LIN {X 0,Y 467.698,Z 216.222,A -85,B 0,C 180,E1 -7463.962,E2 -7463.962} C_VEL
LIN {X 0,Y 467.802,Z 216.212,A -85,B 0,C 180,E1 -7467.417,E2 -7467.417} C_VEL
LIN {X 0,Y 467.814,Z 216.207,A -85,B 0,C 180,E1 -7470,E2 -7470} C_VEL
LIN {X 0,Y 467.802,Z 216.211,A -85,B 0,C 180,E1 -7472.583,E2 -7472.583} C_VEL
LIN {X 0,Y 467.698,Z 216.222,A -85,B 0,C 180,E1 -7476.038,E2 -7476.038} C_VEL
LIN {X 0,Y 467.633,Z 216.235,A -85,B 0,C 180,E1 -7478.643,E2 -7478.643} C_VEL
LIN {X 0,Y 467.672,Z 216.264,A -85,B 0,C 180,E1 -7482.09,E2 -7482.09} C_VEL
LIN {X 0,Y 468.717,Z 223.503,A -85,B 0,C 180,E1 -7483.659,E2 -7483.659} C_VEL
LIN {X 0,Y 468.443,Z 235.17,A -85,B 0,C 180,E1 -7486.063,E2 -7486.063} C_VEL
LIN {X 0,Y 471.362,Z 250.846,A -85,B 0,C 180,E1 -7486.427,E2 -7486.427} C_VEL
LIN {X 0,Y 470.517,Z 341.953,A -85,B 0,C 180,E1 -7487.858,E2 -7487.858} C_VEL
LIN {X 0,Y 470.242,Z 355.17,A -85,B 0,C 180,E1 -7488.235,E2 -7488.235} C_VEL
LIN {X 0,Y 469.903,Z 367.496,A -85,B 0,C 180,E1 -7488.757,E2 -7488.757} C_VEL
LIN {X 0,Y 469.518,Z 379.697,A -85,B 0,C 180,E1 -7489.46,E2 -7489.46} C_VEL
LIN {X 0,Y 469.025,Z 390.638,A -85,B 0,C 180,E1 -7490.273,E2 -7490.273} C_VEL
LIN {X 0,Y 468.536,Z 401.021,A -85,B 0,C 180,E1 -7491.237,E2 -7491.237} C_VEL
LIN {X 0,Y 468.092,Z 410.16,A -85,B 0,C 180,E1 -7492.278,E2 -7492.278} C_VEL
LIN {X 0,Y 467.664,Z 419.305,A -85,B 0,C 180,E1 -7493.572,E2 -7493.572} C_VEL
LIN {X 0,Y 467.295,Z 426.861,A -85,B 0,C 180,E1 -7494.904,E2 -7494.904} C_VEL
LIN {X 0,Y 467.014,Z 433.368,A -85,B 0,C 180,E1 -7496.355,E2 -7496.355} C_VEL
LIN {X 0,Y 466.823,Z 438.356,A -85,B 0,C 180,E1 -7497.82,E2 -7497.82} C_VEL
LIN {X 0,Y 466.725,Z 441.75,A -85,B 0,C 180,E1 -7499.163,E2 -7499.163} C_VEL
LIN {X 0,Y 466.568,Z 444.553,A -85,B 0,C 180,E1 -7500.855,E2 -7500.855} C_VEL
LIN {X 0,Y 466.525,Z 445.764,A -85,B 0,C 180,E1 -7502.491,E2 -7502.491} C_VEL
LIN {X 0,Y 466.515,Z 445.58,A -85,B 0,C 180,E1 -7504.062,E2 -7504.062} C_VEL
LIN {X 0,Y 466.566,Z 444.162,A -85,B 0,C 180,E1 -7505.582,E2 -7505.582} C_VEL
LIN {X 0,Y 466.714,Z 441.569,A -85,B 0,C 180,E1 -7507.064,E2 -7507.064} C_VEL
LIN {X 0,Y 466.883,Z 437.838,A -85,B 0,C 180,E1 -7508.498,E2 -7508.498} C_VEL
LIN {X 0,Y 467.075,Z 432.923,A -85,B 0,C 180,E1 -7509.892,E2 -7509.892} C_VEL
LIN {X 0,Y 467.372,Z 425.882,A -85,B 0,C 180,E1 -7511.424,E2 -7511.424} C_VEL
LIN {X 0,Y 467.654,Z 419.182,A -85,B 0,C 180,E1 -7512.587,E2 -7512.587} C_VEL
LIN {X 0,Y 468.1,Z 411.54,A -85,B 0,C 180,E1 -7513.679,E2 -7513.679} C_VEL
LIN {X 0,Y 468.582,Z 401.758,A -85,B 0,C 180,E1 -7514.822,E2 -7514.822} C_VEL
LIN {X 0,Y 469.08,Z 390.527,A -85,B 0,C 180,E1 -7515.87,E2 -7515.87} C_VEL
LIN {X 0,Y 469.594,Z 379.793,A -85,B 0,C 180,E1 -7516.666,E2 -7516.666} C_VEL
LIN {X 0,Y 470.011,Z 367.432,A -85,B 0,C 180,E1 -7517.375,E2 -7517.375} C_VEL
LIN {X 0,Y 470.382,Z 354.341,A -85,B 0,C 180,E1 -7517.921,E2 -7517.921} C_VEL
LIN {X 0,Y 470.62,Z 341.699,A -85,B 0,C 180,E1 -7518.271,E2 -7518.271} C_VEL
LIN {X 0,Y 471.439,Z 249.982,A -85,B 0,C 180,E1 -7519.719,E2 -7519.719} C_VEL
LIN {X 0,Y 468.517,Z 235.14,A -85,B 0,C 180,E1 -7520.078,E2 -7520.078} C_VEL
LIN {X 0,Y 468.684,Z 222.897,A -85,B 0,C 180,E1 -7522.429,E2 -7522.429} C_VEL
LIN {X 0,Y 467.576,Z 216.244,A -85,B 0,C 180,E1 -7523.788,E2 -7523.788} C_VEL
LIN {X 0,Y 467.548,Z 216.245,A -85,B 0,C 180,E1 -7526.217,E2 -7526.217} C_VEL
LIN {X 0,Y 467.538,Z 216.249,A -85,B 0,C 180,E1 -7529.272,E2 -7529.272} C_VEL
LIN {X 0,Y 467.611,Z 216.236,A -85,B 0,C 180,E1 -7532.464,E2 -7532.464} C_VEL
LIN {X 0,Y 467.572,Z 216.245,A -85,B 0,C 180,E1 -7535.118,E2 -7535.118} C_VEL
LIN {X 0,Y 467.505,Z 216.247,A -85,B 0,C 180,E1 -7537.931,E2 -7537.931} C_VEL
LIN {X 0,Y 467.596,Z 216.24,A -85,B 0,C 180,E1 -7540.697,E2 -7540.697} C_VEL
LIN {X 0,Y 467.625,Z 216.234,A -85,B 0,C 180,E1 -7544.12,E2 -7544.12} C_VEL
LIN {X 0,Y 467.662,Z 216.227,A -85,B 0,C 180,E1 -7547.86,E2 -7547.86} C_VEL
LIN {X 0,Y 467.652,Z 216.229,A -85,B 0,C 180,E1 -7551.362,E2 -7551.362} C_VEL
LIN {X 0,Y 467.713,Z 216.221,A -85,B 0,C 180,E1 -7553.967,E2 -7553.967} C_VEL
LIN {X 0,Y 467.841,Z 216.204,A -85,B 0,C 180,E1 -7557.422,E2 -7557.422} C_VEL
LIN {X 0,Y 467.865,Z 216.202,A -85,B 0,C 180,E1 -7560.005,E2 -7560.005} C_VEL
LIN {X 0,Y 467.809,Z 216.211,A -85,B 0,C 180,E1 -7562.588,E2 -7562.588} C_VEL
LIN {X 0,Y 467.713,Z 216.218,A -85,B 0,C 180,E1 -7566.042,E2 -7566.042} C_VEL
LIN {X 0,Y 467.653,Z 216.234,A -85,B 0,C 180,E1 -7568.648,E2 -7568.648} C_VEL
LIN {X 0,Y 467.65,Z 216.23,A -85,B 0,C 180,E1 -7572.15,E2 -7572.15} C_VEL
LIN {X 0,Y 467.635,Z 216.23,A -85,B 0,C 180,E1 -7575.699,E2 -7575.699} C_VEL
LIN {X 0,Y 467.619,Z 216.232,A -85,B 0,C 180,E1 -7579.312,E2 -7579.312} C_VEL
LIN {X 0,Y 467.53,Z 216.244,A -85,B 0,C 180,E1 -7582.078,E2 -7582.078} C_VEL
LIN {X 0,Y 467.549,Z 216.243,A -85,B 0,C 180,E1 -7584.894,E2 -7584.894} C_VEL
LIN {X 0,Y 467.547,Z 216.241,A -85,B 0,C 180,E1 -7587.777,E2 -7587.777} C_VEL
LIN {X 0,Y 467.548,Z 216.243,A -85,B 0,C 180,E1 -7591.043,E2 -7591.043} C_VEL
LIN {X 0,Y 467.578,Z 216.24,A -85,B 0,C 180,E1 -7594.243,E2 -7594.243} C_VEL
LIN {X 0,Y 467.517,Z 216.245,A -85,B 0,C 180,E1 -7597.183,E2 -7597.183} C_VEL
LIN {X 0,Y 467.522,Z 216.249,A -85,B 0,C 180,E1 -7600.274,E2 -7600.274} C_VEL
LIN {X 0,Y 467.522,Z 216.251,A -85,B 0,C 180,E1 -7602.571,E2 -7602.571} C_VEL
LIN {X 0,Y 467.558,Z 216.243,A -85,B 0,C 180,E1 -7605.053,E2 -7605.053} C_VEL
LIN {X 0,Y 467.556,Z 216.244,A -85,B 0,C 180,E1 -7608.73,E2 -7608.73} C_VEL
LIN {X 0,Y 467.539,Z 216.247,A -85,B 0,C 180,E1 -7611.954,E2 -7611.954} C_VEL
LIN {X 0,Y 467.545,Z 216.243,A -85,B 0,C 180,E1 -7615.167,E2 -7615.167} C_VEL
LIN {X 0,Y 467.549,Z 216.252,A -85,B 0,C 180,E1 -7618.258,E2 -7618.258} C_VEL
LIN {X 0,Y 467.526,Z 216.249,A -85,B 0,C 180,E1 -7621.248,E2 -7621.248} C_VEL
LIN {X 0,Y 467.563,Z 216.308,A -85,B 0,C 180,E1 -7624.098,E2 -7624.098} C_VEL
LIN {X 0,Y 469.703,Z 227.399,A -85,B 0,C 180,E1 -7626.173,E2 -7626.173} C_VEL
LIN {X 0,Y 469.196,Z 242.28,A -85,B 0,C 180,E1 -7628.742,E2 -7628.742} C_VEL
LIN {X 0,Y 468.518,Z 260.61,A -85,B 0,C 180,E1 -7631.865,E2 -7631.865} C_VEL
LIN {X 0,Y 468.314,Z 267.311,A -85,B 0,C 180,E1 -7632.96,E2 -7632.96} C_VEL
LIN {X 0,Y 471.186,Z 286.372,A -85,B 0,C 180,E1 -7633.375,E2 -7633.375} C_VEL
LIN {X 0,Y 470.504,Z 375.82,A -85,B 0,C 180,E1 -7634.792,E2 -7634.792} C_VEL
LIN {X 0,Y 470.072,Z 389.744,A -85,B 0,C 180,E1 -7635.193,E2 -7635.193} C_VEL
LIN {X 0,Y 469.595,Z 402.758,A -85,B 0,C 180,E1 -7635.759,E2 -7635.759} C_VEL
LIN {X 0,Y 469.093,Z 414.583,A -85,B 0,C 180,E1 -7636.462,E2 -7636.462} C_VEL
LIN {X 0,Y 468.57,Z 426.698,A -85,B 0,C 180,E1 -7637.389,E2 -7637.389} C_VEL
LIN {X 0,Y 468.149,Z 436.288,A -85,B 0,C 180,E1 -7638.307,E2 -7638.307} C_VEL
LIN {X 0,Y 467.672,Z 445.54,A -85,B 0,C 180,E1 -7639.392,E2 -7639.392} C_VEL
LIN {X 0,Y 467.253,Z 454.552,A -85,B 0,C 180,E1 -7640.695,E2 -7640.695} C_VEL
LIN {X 0,Y 467.003,Z 461.815,A -85,B 0,C 180,E1 -7641.998,E2 -7641.998} C_VEL
LIN {X 0,Y 466.839,Z 466.717,A -85,B 0,C 180,E1 -7643.083,E2 -7643.083} C_VEL
LIN {X 0,Y 466.736,Z 471.485,A -85,B 0,C 180,E1 -7644.383,E2 -7644.383} C_VEL
LIN {X 0,Y 466.649,Z 475.131,A -85,B 0,C 180,E1 -7645.682,E2 -7645.682} C_VEL
LIN {X 0,Y 466.693,Z 477.016,A -85,B 0,C 180,E1 -7646.547,E2 -7646.547} C_VEL
LIN {X 0,Y 466.666,Z 478.428,A -85,B 0,C 180,E1 -7647.411,E2 -7647.411} C_VEL
LIN {X 0,Y 466.624,Z 480.056,A -85,B 0,C 180,E1 -7649.137,E2 -7649.137} C_VEL
LIN {X 0,Y 466.606,Z 480.277,A -85,B 0,C 180,E1 -7650,E2 -7650} C_VEL
LIN {X 0,Y 466.624,Z 480.063,A -85,B 0,C 180,E1 -7650.863,E2 -7650.863} C_VEL
LIN {X 0,Y 466.666,Z 478.457,A -85,B 0,C 180,E1 -7652.589,E2 -7652.589} C_VEL
LIN {X 0,Y 466.693,Z 477.051,A -85,B 0,C 180,E1 -7653.453,E2 -7653.453} C_VEL
LIN {X 0,Y 466.691,Z 474.094,A -85,B 0,C 180,E1 -7654.751,E2 -7654.751} C_VEL
LIN {X 0,Y 466.747,Z 470.089,A -85,B 0,C 180,E1 -7656.05,E2 -7656.05} C_VEL
LIN {X 0,Y 466.926,Z 463.923,A -85,B 0,C 180,E1 -7657.568,E2 -7657.568} C_VEL
LIN {X 0,Y 467.166,Z 457.189,A -85,B 0,C 180,E1 -7658.87,E2 -7658.87} C_VEL
LIN {X 0,Y 467.493,Z 448.832,A -85,B 0,C 180,E1 -7660.174,E2 -7660.174} C_VEL
LIN {X 0,Y 467.955,Z 440.241,A -85,B 0,C 180,E1 -7661.259,E2 -7661.259} C_VEL
LIN {X 0,Y 468.445,Z 430.165,A -85,B 0,C 180,E1 -7662.295,E2 -7662.295} C_VEL
LIN {X 0,Y 468.881,Z 419.128,A -85,B 0,C 180,E1 -7663.213,E2 -7663.213} C_VEL
LIN {X 0,Y 469.377,Z 407.552,A -85,B 0,C 180,E1 -7663.971,E2 -7663.971} C_VEL
LIN {X 0,Y 469.837,Z 395.543,A -85,B 0,C 180,E1 -7664.565,E2 -7664.565} C_VEL
LIN {X 0,Y 470.253,Z 382.567,A -85,B 0,C 180,E1 -7665.023,E2 -7665.023} C_VEL
LIN {X 0,Y 470.538,Z 368.731,A -85,B 0,C 180,E1 -7665.318,E2 -7665.318} C_VEL
LIN {X 0,Y 471.01,Z 285.555,A -85,B 0,C 180,E1 -7666.617,E2 -7666.617} C_VEL
LIN {X 0,Y 468.273,Z 267.515,A -85,B 0,C 180,E1 -7667.017,E2 -7667.017} C_VEL
LIN {X 0,Y 468.932,Z 250.577,A -85,B 0,C 180,E1 -7669.935,E2 -7669.935} C_VEL
LIN {X 0,Y 469.674,Z 234.928,A -85,B 0,C 180,E1 -7672.663,E2 -7672.663} C_VEL
LIN {X 0,Y 469.875,Z 228.39,A -85,B 0,C 180,E1 -7673.818,E2 -7673.818} C_VEL
LIN {X 0,Y 467.555,Z 216.246,A -85,B 0,C 180,E1 -7676.142,E2 -7676.142} C_VEL
LIN {X 0,Y 467.532,Z 216.249,A -85,B 0,C 180,E1 -7679.32,E2 -7679.32} C_VEL
LIN {X 0,Y 467.545,Z 216.248,A -85,B 0,C 180,E1 -7681.742,E2 -7681.742} C_VEL
LIN {X 0,Y 467.518,Z 216.244,A -85,B 0,C 180,E1 -7684.836,E2 -7684.836} C_VEL
LIN {X 0,Y 467.537,Z 216.246,A -85,B 0,C 180,E1 -7688.046,E2 -7688.046} C_VEL
LIN {X 0,Y 467.553,Z 216.243,A -85,B 0,C 180,E1 -7691.404,E2 -7691.404} C_VEL
LIN {X 0,Y 467.535,Z 216.243,A -85,B 0,C 180,E1 -7695.045,E2 -7695.045} C_VEL
LIN {X 0,Y 467.554,Z 216.24,A -85,B 0,C 180,E1 -7698.591,E2 -7698.591} C_VEL
LIN {X 0,Y 467.533,Z 216.247,A -85,B 0,C 180,E1 -7701.949,E2 -7701.949} C_VEL
LIN {X 0,Y 467.518,Z 216.246,A -85,B 0,C 180,E1 -7705.16,E2 -7705.16} C_VEL
LIN {X 0,Y 467.544,Z 216.242,A -85,B 0,C 180,E1 -7708.253,E2 -7708.253} C_VEL
LIN {X 0,Y 467.52,Z 216.247,A -85,B 0,C 180,E1 -7711.243,E2 -7711.243} C_VEL
LIN {X 0,Y 467.558,Z 216.24,A -85,B 0,C 180,E1 -7714.403,E2 -7714.403} C_VEL
LIN {X 0,Y 467.571,Z 216.239,A -85,B 0,C 180,E1 -7716.992,E2 -7716.992} C_VEL
LIN {X 0,Y 467.589,Z 216.241,A -85,B 0,C 180,E1 -7719.772,E2 -7719.772} C_VEL
LIN {X 0,Y 467.568,Z 216.238,A -85,B 0,C 180,E1 -7722.501,E2 -7722.501} C_VEL
LIN {X 0,Y 467.589,Z 216.238,A -85,B 0,C 180,E1 -7725.192,E2 -7725.192} C_VEL
LIN {X 0,Y 467.629,Z 216.235,A -85,B 0,C 180,E1 -7727.85,E2 -7727.85} C_VEL
LIN {X 0,Y 467.621,Z 216.237,A -85,B 0,C 180,E1 -7731.352,E2 -7731.352} C_VEL
LIN {X 0,Y 467.692,Z 216.225,A -85,B 0,C 180,E1 -7733.957,E2 -7733.957} C_VEL
LIN {X 0,Y 467.777,Z 216.219,A -85,B 0,C 180,E1 -7737.412,E2 -7737.412} C_VEL
LIN {X 0,Y 467.833,Z 216.207,A -85,B 0,C 180,E1 -7739.995,E2 -7739.995} C_VEL
LIN {X 0,Y 467.806,Z 216.208,A -85,B 0,C 180,E1 -7742.578,E2 -7742.578} C_VEL
LIN {X 0,Y 467.675,Z 216.226,A -85,B 0,C 180,E1 -7746.033,E2 -7746.033} C_VEL
LIN {X 0,Y 467.616,Z 216.232,A -85,B 0,C 180,E1 -7748.639,E2 -7748.639} C_VEL
LIN {X 0,Y 467.634,Z 216.23,A -85,B 0,C 180,E1 -7752.14,E2 -7752.14} C_VEL
LIN {X 0,Y 467.624,Z 216.233,A -85,B 0,C 180,E1 -7755.879,E2 -7755.879} C_VEL
LIN {X 0,Y 467.594,Z 216.242,A -85,B 0,C 180,E1 -7759.303,E2 -7759.303} C_VEL
LIN {X 0,Y 467.501,Z 216.247,A -85,B 0,C 180,E1 -7762.069,E2 -7762.069} C_VEL
LIN {X 0,Y 467.536,Z 216.244,A -85,B 0,C 180,E1 -7764.884,E2 -7764.884} C_VEL
LIN {X 0,Y 467.581,Z 216.239,A -85,B 0,C 180,E1 -7767.764,E2 -7767.764} C_VEL
LIN {X 0,Y 467.53,Z 216.247,A -85,B 0,C 180,E1 -7771.039,E2 -7771.039} C_VEL
LIN {X 0,Y 467.548,Z 216.24,A -85,B 0,C 180,E1 -7774.237,E2 -7774.237} C_VEL
LIN {X 0,Y 467.505,Z 216.252,A -85,B 0,C 180,E1 -7777.181,E2 -7777.181} C_VEL
LIN {X 0,Y 467.533,Z 216.242,A -85,B 0,C 180,E1 -7780.26,E2 -7780.26} C_VEL
LIN {X 0,Y 467.541,Z 216.242,A -85,B 0,C 180,E1 -7782.562,E2 -7782.562} C_VEL
LIN {X 0,Y 467.522,Z 216.249,A -85,B 0,C 180,E1 -7785.049,E2 -7785.049} C_VEL
LIN {X 0,Y 467.539,Z 216.247,A -85,B 0,C 180,E1 -7787.436,E2 -7787.436} C_VEL
LIN {X 0,Y 467.53,Z 216.246,A -85,B 0,C 180,E1 -7790.851,E2 -7790.851} C_VEL
LIN {X 0,Y 467.51,Z 216.245,A -85,B 0,C 180,E1 -7794.256,E2 -7794.256} C_VEL
LIN {X 0,Y 467.526,Z 216.25,A -85,B 0,C 180,E1 -7797.317,E2 -7797.317} C_VEL
LIN {X 0,Y 467.519,Z 216.246,A -85,B 0,C 180,E1 -7800.663,E2 -7800.663} C_VEL
LIN {X 0,Y 467.561,Z 216.247,A -85,B 0,C 180,E1 -7803.197,E2 -7803.197} C_VEL
LIN {X 0,Y 467.526,Z 216.243,A -85,B 0,C 180,E1 -7806.055,E2 -7806.055} C_VEL
LIN {X 0,Y 467.579,Z 216.241,A -85,B 0,C 180,E1 -7808.855,E2 -7808.855} C_VEL
LIN {X 0,Y 467.578,Z 216.239,A -85,B 0,C 180,E1 -7811.613,E2 -7811.613} C_VEL
LIN {X 0,Y 467.591,Z 216.235,A -85,B 0,C 180,E1 -7814.304,E2 -7814.304} C_VEL
LIN {X 0,Y 467.536,Z 216.247,A -85,B 0,C 180,E1 -7815.371,E2 -7815.371} C_VEL
LIN {X 0,Y 466.869,Z 216.326,A -85,B 0,C 180,E1 -7816.091,E2 -7816.091} C_VEL
LIN {X 0,Y 464.039,Z 216.684,A -85,B 0,C 180,E1 -7817.26,E2 -7817.26} C_VEL
LIN {X 0,Y 461.647,Z 216.978,A -85,B 0,C 180,E1 -7818.203,E2 -7818.203} C_VEL
LIN {X 0,Y 460.618,Z 217.11,A -85,B 0,C 180,E1 -7818.931,E2 -7818.931} C_VEL
LIN {X 0,Y 460.533,Z 217.116,A -85,B 0,C 180,E1 -7819.177,E2 -7819.177} C_VEL
LIN {X 0,Y 460.665,Z 217.1,A -85,B 0,C 180,E1 -7822.527,E2 -7822.527} C_VEL
LIN {X 0,Y 460.644,Z 217.104,A -85,B 0,C 180,E1 -7824.748,E2 -7824.748} C_VEL
LIN {X 0,Y 460.768,Z 217.089,A -85,B 0,C 180,E1 -7827.377,E2 -7827.377} C_VEL
LIN {X 0,Y 460.786,Z 217.083,A -85,B 0,C 180,E1 -7830,E2 -7830} C_VEL
LIN {X 0,Y 460.768,Z 217.088,A -85,B 0,C 180,E1 -7832.623,E2 -7832.623} C_VEL
LIN {X 0,Y 460.664,Z 217.098,A -85,B 0,C 180,E1 -7836.13,E2 -7836.13} C_VEL
LIN {X 0,Y 460.6,Z 217.113,A -85,B 0,C 180,E1 -7838.776,E2 -7838.776} C_VEL
LIN {X 0,Y 460.656,Z 217.258,A -85,B 0,C 180,E1 -7841.941,E2 -7841.941} C_VEL
LIN {X 0,Y 461.758,Z 225.024,A -85,B 0,C 180,E1 -7843.645,E2 -7843.645} C_VEL
LIN {X 0,Y 461.495,Z 235.327,A -85,B 0,C 180,E1 -7845.796,E2 -7845.796} C_VEL
LIN {X 0,Y 464.529,Z 250.64,A -85,B 0,C 180,E1 -7846.175,E2 -7846.175} C_VEL
LIN {X 0,Y 463.66,Z 342.57,A -85,B 0,C 180,E1 -7847.647,E2 -7847.647} C_VEL
LIN {X 0,Y 463.364,Z 355.678,A -85,B 0,C 180,E1 -7848.029,E2 -7848.029} C_VEL
LIN {X 0,Y 463.007,Z 368.52,A -85,B 0,C 180,E1 -7848.587,E2 -7848.587} C_VEL
LIN {X 0,Y 462.595,Z 380.416,A -85,B 0,C 180,E1 -7849.295,E2 -7849.295} C_VEL
LIN {X 0,Y 462.023,Z 392.472,A -85,B 0,C 180,E1 -7850.223,E2 -7850.223} C_VEL
LIN {X 0,Y 461.497,Z 402.613,A -85,B 0,C 180,E1 -7851.203,E2 -7851.203} C_VEL
LIN {X 0,Y 460.961,Z 412.559,A -85,B 0,C 180,E1 -7852.405,E2 -7852.405} C_VEL
LIN {X 0,Y 460.527,Z 421.341,A -85,B 0,C 180,E1 -7853.723,E2 -7853.723} C_VEL
LIN {X 0,Y 460.239,Z 428.51,A -85,B 0,C 180,E1 -7855.071,E2 -7855.071} C_VEL
LIN {X 0,Y 459.943,Z 433.788,A -85,B 0,C 180,E1 -7856.303,E2 -7856.303} C_VEL
LIN {X 0,Y 459.789,Z 438.129,A -85,B 0,C 180,E1 -7857.575,E2 -7857.575} C_VEL
LIN {X 0,Y 459.676,Z 441.325,A -85,B 0,C 180,E1 -7858.789,E2 -7858.789} C_VEL
LIN {X 0,Y 459.5,Z 444.151,A -85,B 0,C 180,E1 -7860.313,E2 -7860.313} C_VEL
LIN {X 0,Y 459.457,Z 445.324,A -85,B 0,C 180,E1 -7861.336,E2 -7861.336} C_VEL
LIN {X 0,Y 459.411,Z 446.073,A -85,B 0,C 180,E1 -7862.728,E2 -7862.728} C_VEL
LIN {X 0,Y 459.432,Z 445.628,A -85,B 0,C 180,E1 -7864.47,E2 -7864.47} C_VEL
LIN {X 0,Y 459.511,Z 444.126,A -85,B 0,C 180,E1 -7865.858,E2 -7865.858} C_VEL
LIN {X 0,Y 459.672,Z 441.336,A -85,B 0,C 180,E1 -7867.354,E2 -7867.354} C_VEL
LIN {X 0,Y 459.838,Z 437.42,A -85,B 0,C 180,E1 -7868.801,E2 -7868.801} C_VEL
LIN {X 0,Y 460.069,Z 432.327,A -85,B 0,C 180,E1 -7870.211,E2 -7870.211} C_VEL
LIN {X 0,Y 460.348,Z 425.988,A -85,B 0,C 180,E1 -7871.588,E2 -7871.588} C_VEL
LIN {X 0,Y 460.75,Z 418.144,A -85,B 0,C 180,E1 -7872.943,E2 -7872.943} C_VEL
LIN {X 0,Y 461.204,Z 409.879,A -85,B 0,C 180,E1 -7874.094,E2 -7874.094} C_VEL
LIN {X 0,Y 461.732,Z 400.209,A -85,B 0,C 180,E1 -7875.193,E2 -7875.193} C_VEL
LIN {X 0,Y 462.192,Z 390.615,A -85,B 0,C 180,E1 -7876.084,E2 -7876.084} C_VEL
LIN {X 0,Y 462.707,Z 379.833,A -85,B 0,C 180,E1 -7876.892,E2 -7876.892} C_VEL
LIN {X 0,Y 463.142,Z 367.848,A -85,B 0,C 180,E1 -7877.588,E2 -7877.588} C_VEL
LIN {X 0,Y 463.542,Z 354.862,A -85,B 0,C 180,E1 -7878.14,E2 -7878.14} C_VEL
LIN {X 0,Y 463.798,Z 341.73,A -85,B 0,C 180,E1 -7878.509,E2 -7878.509} C_VEL
LIN {X 0,Y 464.545,Z 250.039,A -85,B 0,C 180,E1 -7879.985,E2 -7879.985} C_VEL
LIN {X 0,Y 461.585,Z 235.343,A -85,B 0,C 180,E1 -7880.362,E2 -7880.362} C_VEL
LIN {X 0,Y 461.766,Z 224.266,A -85,B 0,C 180,E1 -7882.507,E2 -7882.507} C_VEL
LIN {X 0,Y 460.526,Z 217.122,A -85,B 0,C 180,E1 -7883.979,E2 -7883.979} C_VEL
LIN {X 0,Y 460.493,Z 217.128,A -85,B 0,C 180,E1 -7887.075,E2 -7887.075} C_VEL
LIN {X 0,Y 460.512,Z 217.122,A -85,B 0,C 180,E1 -7890.443,E2 -7890.443} C_VEL
LIN {X 0,Y 460.551,Z 217.118,A -85,B 0,C 180,E1 -7892.762,E2 -7892.762} C_VEL
LIN {X 0,Y 460.511,Z 217.12,A -85,B 0,C 180,E1 -7895.673,E2 -7895.673} C_VEL
LIN {X 0,Y 460.493,Z 217.124,A -85,B 0,C 180,E1 -7898.584,E2 -7898.584} C_VEL
LIN {X 0,Y 460.564,Z 217.117,A -85,B 0,C 180,E1 -7901.316,E2 -7901.316} C_VEL
LIN {X 0,Y 460.58,Z 217.111,A -85,B 0,C 180,E1 -7904.064,E2 -7904.064} C_VEL
LIN {X 0,Y 460.609,Z 217.106,A -85,B 0,C 180,E1 -7907.672,E2 -7907.672} C_VEL
LIN {X 0,Y 460.603,Z 217.108,A -85,B 0,C 180,E1 -7911.229,E2 -7911.229} C_VEL
LIN {X 0,Y 460.679,Z 217.097,A -85,B 0,C 180,E1 -7913.875,E2 -7913.875} C_VEL
LIN {X 0,Y 460.783,Z 217.084,A -85,B 0,C 180,E1 -7917.383,E2 -7917.383} C_VEL
LIN {X 0,Y 460.835,Z 217.078,A -85,B 0,C 180,E1 -7920.005,E2 -7920.005} C_VEL
LIN {X 0,Y 460.753,Z 217.09,A -85,B 0,C 180,E1 -7922.628,E2 -7922.628} C_VEL
LIN {X 0,Y 460.679,Z 217.095,A -85,B 0,C 180,E1 -7926.135,E2 -7926.135} C_VEL
LIN {X 0,Y 460.601,Z 217.11,A -85,B 0,C 180,E1 -7928.781,E2 -7928.781} C_VEL
LIN {X 0,Y 460.592,Z 217.113,A -85,B 0,C 180,E1 -7932.439,E2 -7932.439} C_VEL
LIN {X 0,Y 460.598,Z 217.108,A -85,B 0,C 180,E1 -7936.002,E2 -7936.002} C_VEL
LIN {X 0,Y 460.566,Z 217.11,A -85,B 0,C 180,E1 -7939.62,E2 -7939.62} C_VEL
LIN {X 0,Y 460.507,Z 217.121,A -85,B 0,C 180,E1 -7942.433,E2 -7942.433} C_VEL
LIN {X 0,Y 460.522,Z 217.116,A -85,B 0,C 180,E1 -7945.793,E2 -7945.793} C_VEL
LIN {X 0,Y 460.525,Z 217.115,A -85,B 0,C 180,E1 -7949.236,E2 -7949.236} C_VEL
LIN {X 0,Y 460.52,Z 217.122,A -85,B 0,C 180,E1 -7952.289,E2 -7952.289} C_VEL
LIN {X 0,Y 460.503,Z 217.119,A -85,B 0,C 180,E1 -7955.45,E2 -7955.45} C_VEL
LIN {X 0,Y 460.486,Z 217.123,A -85,B 0,C 180,E1 -7958.89,E2 -7958.89} C_VEL
LIN {X 0,Y 460.5,Z 217.121,A -85,B 0,C 180,E1 -7961.6,E2 -7961.6} C_VEL
LIN {X 0,Y 460.511,Z 217.124,A -85,B 0,C 180,E1 -7964.593,E2 -7964.593} C_VEL
LIN {X 0,Y 460.477,Z 217.126,A -85,B 0,C 180,E1 -7967.815,E2 -7967.815} C_VEL
LIN {X 0,Y 460.48,Z 217.129,A -85,B 0,C 180,E1 -7970.134,E2 -7970.134} C_VEL
LIN {X 0,Y 460.46,Z 217.126,A -85,B 0,C 180,E1 -7973.47,E2 -7973.47} C_VEL
LIN {X 0,Y 460.506,Z 217.124,A -85,B 0,C 180,E1 -7976.674,E2 -7976.674} C_VEL
LIN {X 0,Y 460.485,Z 217.129,A -85,B 0,C 180,E1 -7979.759,E2 -7979.759} C_VEL
LIN {X 0,Y 460.484,Z 217.126,A -85,B 0,C 180,E1 -7982.751,E2 -7982.751} C_VEL
LIN {X 0,Y 460.511,Z 217.136,A -85,B 0,C 180,E1 -7983.867,E2 -7983.867} C_VEL
LIN {X 0,Y 462.61,Z 227.87,A -85,B 0,C 180,E1 -7985.913,E2 -7985.913} C_VEL
LIN {X 0,Y 462.708,Z 232.485,A -85,B 0,C 180,E1 -7986.74,E2 -7986.74} C_VEL
LIN {X 0,Y 461.993,Z 248.444,A -85,B 0,C 180,E1 -7989.52,E2 -7989.52} C_VEL
LIN {X 0,Y 461.402,Z 264.339,A -85,B 0,C 180,E1 -7992.264,E2 -7992.264} C_VEL
LIN {X 0,Y 461.317,Z 266.734,A -85,B 0,C 180,E1 -7992.675,E2 -7992.675} C_VEL
LIN {X 0,Y 464.405,Z 287.188,A -85,B 0,C 180,E1 -7993.134,E2 -7993.134} C_VEL
LIN {X 0,Y 463.679,Z 375.696,A -85,B 0,C 180,E1 -7994.562,E2 -7994.562} C_VEL
LIN {X 0,Y 463.213,Z 389.565,A -85,B 0,C 180,E1 -7994.969,E2 -7994.969} C_VEL
LIN {X 0,Y 462.72,Z 402.546,A -85,B 0,C 180,E1 -7995.543,E2 -7995.543} C_VEL
LIN {X 0,Y 462.157,Z 414.355,A -85,B 0,C 180,E1 -7996.255,E2 -7996.255} C_VEL
LIN {X 0,Y 461.664,Z 425.832,A -85,B 0,C 180,E1 -7997.143,E2 -7997.143} C_VEL
LIN {X 0,Y 461.176,Z 436.039,A -85,B 0,C 180,E1 -7998.128,E2 -7998.128} C_VEL
LIN {X 0,Y 460.643,Z 445.284,A -85,B 0,C 180,E1 -7999.229,E2 -7999.229} C_VEL
LIN {X 0,Y 460.206,Z 454.294,A -85,B 0,C 180,E1 -8000.551,E2 -8000.551} C_VEL
LIN {X 0,Y 459.931,Z 461.556,A -85,B 0,C 180,E1 -8001.875,E2 -8001.875} C_VEL
LIN {X 0,Y 459.745,Z 467.64,A -85,B 0,C 180,E1 -8003.273,E2 -8003.273} C_VEL
LIN {X 0,Y 459.646,Z 472.554,A -85,B 0,C 180,E1 -8004.736,E2 -8004.736} C_VEL
LIN {X 0,Y 459.567,Z 474.873,A -85,B 0,C 180,E1 -8005.615,E2 -8005.615} C_VEL
LIN {X 0,Y 459.588,Z 476.756,A -85,B 0,C 180,E1 -8006.493,E2 -8006.493} C_VEL
LIN {X 0,Y 459.588,Z 478.169,A -85,B 0,C 180,E1 -8007.371,E2 -8007.371} C_VEL
LIN {X 0,Y 459.528,Z 479.795,A -85,B 0,C 180,E1 -8009.124,E2 -8009.124} C_VEL
LIN {X 0,Y 459.537,Z 480.016,A -85,B 0,C 180,E1 -8010,E2 -8010} C_VEL
LIN {X 0,Y 459.546,Z 479.19,A -85,B 0,C 180,E1 -8011.753,E2 -8011.753} C_VEL
LIN {X 0,Y 459.589,Z 478.191,A -85,B 0,C 180,E1 -8012.629,E2 -8012.629} C_VEL
LIN {X 0,Y 459.589,Z 476.78,A -85,B 0,C 180,E1 -8013.507,E2 -8013.507} C_VEL
LIN {X 0,Y 459.618,Z 473.82,A -85,B 0,C 180,E1 -8014.824,E2 -8014.824} C_VEL
LIN {X 0,Y 459.725,Z 468.764,A -85,B 0,C 180,E1 -8016.431,E2 -8016.431} C_VEL
LIN {X 0,Y 459.894,Z 462.615,A -85,B 0,C 180,E1 -8017.905,E2 -8017.905} C_VEL
LIN {X 0,Y 460.169,Z 455.643,A -85,B 0,C 180,E1 -8019.228,E2 -8019.228} C_VEL
LIN {X 0,Y 460.527,Z 446.899,A -85,B 0,C 180,E1 -8020.552,E2 -8020.552} C_VEL
LIN {X 0,Y 461.051,Z 437.948,A -85,B 0,C 180,E1 -8021.652,E2 -8021.652} C_VEL
LIN {X 0,Y 461.554,Z 427.263,A -85,B 0,C 180,E1 -8022.723,E2 -8022.723} C_VEL
LIN {X 0,Y 462.091,Z 415.709,A -85,B 0,C 180,E1 -8023.635,E2 -8023.635} C_VEL
LIN {X 0,Y 462.606,Z 403.161,A -85,B 0,C 180,E1 -8024.405,E2 -8024.405} C_VEL
LIN {X 0,Y 463.161,Z 390.339,A -85,B 0,C 180,E1 -8024.977,E2 -8024.977} C_VEL
LIN {X 0,Y 463.504,Z 376.681,A -85,B 0,C 180,E1 -8025.387,E2 -8025.387} C_VEL
LIN {X 0,Y 464.105,Z 323.215,A -85,B 0,C 180,E1 -8026.253,E2 -8026.253} C_VEL
LIN {X 0,Y 464.146,Z 285.68,A -85,B 0,C 180,E1 -8026.858,E2 -8026.858} C_VEL
LIN {X 0,Y 461.309,Z 267.29,A -85,B 0,C 180,E1 -8027.271,E2 -8027.271} C_VEL
LIN {X 0,Y 462.003,Z 250.301,A -85,B 0,C 180,E1 -8030.247,E2 -8030.247} C_VEL
LIN {X 0,Y 462.76,Z 234.639,A -85,B 0,C 180,E1 -8033.02,E2 -8033.02} C_VEL
LIN {X 0,Y 462.898,Z 229.408,A -85,B 0,C 180,E1 -8033.962,E2 -8033.962} C_VEL
LIN {X 0,Y 460.511,Z 217.124,A -85,B 0,C 180,E1 -8036.359,E2 -8036.359} C_VEL
LIN {X 0,Y 460.499,Z 217.125,A -85,B 0,C 180,E1 -8039.547,E2 -8039.547} C_VEL
LIN {X 0,Y 460.49,Z 217.122,A -85,B 0,C 180,E1 -8042.287,E2 -8042.287} C_VEL
LIN {X 0,Y 460.466,Z 217.126,A -85,B 0,C 180,E1 -8045.449,E2 -8045.449} C_VEL
LIN {X 0,Y 460.496,Z 217.119,A -85,B 0,C 180,E1 -8048.735,E2 -8048.735} C_VEL
LIN {X 0,Y 460.5,Z 217.124,A -85,B 0,C 180,E1 -8051.594,E2 -8051.594} C_VEL
LIN {X 0,Y 460.481,Z 217.121,A -85,B 0,C 180,E1 -8054.591,E2 -8054.591} C_VEL
LIN {X 0,Y 460.476,Z 217.129,A -85,B 0,C 180,E1 -8057.81,E2 -8057.81} C_VEL
LIN {X 0,Y 460.477,Z 217.124,A -85,B 0,C 180,E1 -8060.128,E2 -8060.128} C_VEL
LIN {X 0,Y 460.473,Z 217.122,A -85,B 0,C 180,E1 -8062.526,E2 -8062.526} C_VEL
LIN {X 0,Y 460.512,Z 217.124,A -85,B 0,C 180,E1 -8065.617,E2 -8065.617} C_VEL
LIN {X 0,Y 460.508,Z 217.117,A -85,B 0,C 180,E1 -8068.739,E2 -8068.739} C_VEL
LIN {X 0,Y 460.493,Z 217.126,A -85,B 0,C 180,E1 -8071.759,E2 -8071.759} C_VEL
LIN {X 0,Y 460.506,Z 217.118,A -85,B 0,C 180,E1 -8074.698,E2 -8074.698} C_VEL
LIN {X 0,Y 460.504,Z 217.125,A -85,B 0,C 180,E1 -8077.567,E2 -8077.567} C_VEL
LIN {X 0,Y 460.518,Z 217.117,A -85,B 0,C 180,E1 -8080.378,E2 -8080.378} C_VEL
LIN {X 0,Y 460.539,Z 217.116,A -85,B 0,C 180,E1 -8083.141,E2 -8083.141} C_VEL
LIN {X 0,Y 460.534,Z 217.119,A -85,B 0,C 180,E1 -8085.863,E2 -8085.863} C_VEL
LIN {X 0,Y 460.573,Z 217.109,A -85,B 0,C 180,E1 -8088.554,E2 -8088.554} C_VEL
LIN {X 0,Y 460.615,Z 217.106,A -85,B 0,C 180,E1 -8092.103,E2 -8092.103} C_VEL
LIN {X 0,Y 460.662,Z 217.098,A -85,B 0,C 180,E1 -8094.743,E2 -8094.743} C_VEL
LIN {X 0,Y 460.7,Z 217.094,A -85,B 0,C 180,E1 -8098.247,E2 -8098.247} C_VEL
LIN {X 0,Y 460.782,Z 217.085,A -85,B 0,C 180,E1 -8099.995,E2 -8099.995} C_VEL
LIN {X 0,Y 460.75,Z 217.087,A -85,B 0,C 180,E1 -8102.618,E2 -8102.618} C_VEL
LIN {X 0,Y 460.642,Z 217.102,A -85,B 0,C 180,E1 -8106.125,E2 -8106.125} C_VEL
LIN {X 0,Y 460.572,Z 217.11,A -85,B 0,C 180,E1 -8108.772,E2 -8108.772} C_VEL
LIN {X 0,Y 460.588,Z 217.108,A -85,B 0,C 180,E1 -8112.329,E2 -8112.329} C_VEL
LIN {X 0,Y 460.577,Z 217.11,A -85,B 0,C 180,E1 -8115.992,E2 -8115.992} C_VEL
LIN {X 0,Y 460.54,Z 217.119,A -85,B 0,C 180,E1 -8119.61,E2 -8119.61} C_VEL
LIN {X 0,Y 460.477,Z 217.121,A -85,B 0,C 180,E1 -8122.424,E2 -8122.424} C_VEL
LIN {X 0,Y 460.513,Z 217.12,A -85,B 0,C 180,E1 -8125.791,E2 -8125.791} C_VEL
LIN {X 0,Y 460.514,Z 217.117,A -85,B 0,C 180,E1 -8128.228,E2 -8128.228} C_VEL
LIN {X 0,Y 460.483,Z 217.128,A -85,B 0,C 180,E1 -8131.277,E2 -8131.277} C_VEL
LIN {X 0,Y 460.491,Z 217.12,A -85,B 0,C 180,E1 -8134.5,E2 -8134.5} C_VEL
LIN {X 0,Y 460.458,Z 217.128,A -85,B 0,C 180,E1 -8137.618,E2 -8137.618} C_VEL
LIN {X 0,Y 460.497,Z 217.119,A -85,B 0,C 180,E1 -8140.265,E2 -8140.265} C_VEL
LIN {X 0,Y 460.461,Z 217.13,A -85,B 0,C 180,E1 -8143.37,E2 -8143.37} C_VEL
LIN {X 0,Y 460.45,Z 217.126,A -85,B 0,C 180,E1 -8146.62,E2 -8146.62} C_VEL
LIN {X 0,Y 460.49,Z 217.122,A -85,B 0,C 180,E1 -8149.726,E2 -8149.726} C_VEL
LIN {X 0,Y 460.475,Z 217.122,A -85,B 0,C 180,E1 -8152.515,E2 -8152.515} C_VEL
LIN {X 0,Y 460.494,Z 217.122,A -85,B 0,C 180,E1 -8155.62,E2 -8155.62} C_VEL
LIN {X 0,Y 460.48,Z 217.123,A -85,B 0,C 180,E1 -8158.741,E2 -8158.741} C_VEL
LIN {X 0,Y 460.53,Z 217.115,A -85,B 0,C 180,E1 -8162.249,E2 -8162.249} C_VEL
LIN {X 0,Y 460.524,Z 217.118,A -85,B 0,C 180,E1 -8164.704,E2 -8164.704} C_VEL
LIN {X 0,Y 460.48,Z 217.124,A -85,B 0,C 180,E1 -8167.57,E2 -8167.57} C_VEL
LIN {X 0,Y 460.509,Z 217.118,A -85,B 0,C 180,E1 -8170.382,E2 -8170.382} C_VEL
LIN {X 0,Y 460.512,Z 217.125,A -85,B 0,C 180,E1 -8173.145,E2 -8173.145} C_VEL
LIN {X 0,Y 460.495,Z 217.119,A -85,B 0,C 180,E1 -8175.866,E2 -8175.866} C_VEL
LIN {X 0,Y 460.574,Z 217.111,A -85,B 0,C 180,E1 -8178.559,E2 -8178.559} C_VEL
LIN {X 0,Y 460.533,Z 217.116,A -85,B 0,C 180,E1 -8179.177,E2 -8179.177} C_VEL
LIN {X 0,Y 459.869,Z 217.203,A -85,B 0,C 180,E1 -8179.907,E2 -8179.907} C_VEL
LIN {X 0,Y 457.051,Z 217.559,A -85,B 0,C 180,E1 -8181.094,E2 -8181.094} C_VEL
LIN {X 0,Y 454.676,Z 217.854,A -85,B 0,C 180,E1 -8182.051,E2 -8182.051} C_VEL
LIN {X 0,Y 453.665,Z 217.976,A -85,B 0,C 180,E1 -8182.79,E2 -8182.79} C_VEL
LIN {X 0,Y 453.587,Z 217.983,A -85,B 0,C 180,E1 -8183.04,E2 -8183.04} C_VEL
LIN {X 0,Y 453.618,Z 217.979,A -85,B 0,C 180,E1 -8184.666,E2 -8184.666} C_VEL
LIN {X 0,Y 453.709,Z 217.969,A -85,B 0,C 180,E1 -8187.337,E2 -8187.337} C_VEL
LIN {X 0,Y 453.757,Z 217.958,A -85,B 0,C 180,E1 -8190,E2 -8190} C_VEL
LIN {X 0,Y 453.709,Z 217.968,A -85,B 0,C 180,E1 -8192.663,E2 -8192.663} C_VEL
LIN {X 0,Y 453.63,Z 217.975,A -85,B 0,C 180,E1 -8196.226,E2 -8196.226} C_VEL
LIN {X 0,Y 453.554,Z 217.992,A -85,B 0,C 180,E1 -8198.914,E2 -8198.914} C_VEL
LIN {X 0,Y 453.589,Z 218.011,A -85,B 0,C 180,E1 -8201.733,E2 -8201.733} C_VEL
LIN {X 0,Y 454.824,Z 226.528,A -85,B 0,C 180,E1 -8203.629,E2 -8203.629} C_VEL
LIN {X 0,Y 454.568,Z 235.839,A -85,B 0,C 180,E1 -8205.554,E2 -8205.554} C_VEL
LIN {X 0,Y 457.766,Z 252.683,A -85,B 0,C 180,E1 -8205.956,E2 -8205.956} C_VEL
LIN {X 0,Y 456.801,Z 343.136,A -85,B 0,C 180,E1 -8207.428,E2 -8207.428} C_VEL
LIN {X 0,Y 456.456,Z 356.935,A -85,B 0,C 180,E1 -8207.845,E2 -8207.845} C_VEL
LIN {X 0,Y 456.096,Z 369.514,A -85,B 0,C 180,E1 -8208.414,E2 -8208.414} C_VEL
LIN {X 0,Y 455.668,Z 381.003,A -85,B 0,C 180,E1 -8209.117,E2 -8209.117} C_VEL
LIN {X 0,Y 455.141,Z 392.044,A -85,B 0,C 180,E1 -8209.976,E2 -8209.976} C_VEL
LIN {X 0,Y 454.593,Z 402.08,A -85,B 0,C 180,E1 -8210.947,E2 -8210.947} C_VEL
LIN {X 0,Y 454.1,Z 411.118,A -85,B 0,C 180,E1 -8212.019,E2 -8212.019} C_VEL
LIN {X 0,Y 453.651,Z 419.66,A -85,B 0,C 180,E1 -8213.268,E2 -8213.268} C_VEL
LIN {X 0,Y 453.204,Z 427.798,A -85,B 0,C 180,E1 -8214.752,E2 -8214.752} C_VEL
LIN {X 0,Y 452.957,Z 432.725,A -85,B 0,C 180,E1 -8215.871,E2 -8215.871} C_VEL
LIN {X 0,Y 452.753,Z 437.626,A -85,B 0,C 180,E1 -8217.252,E2 -8217.252} C_VEL
LIN {X 0,Y 452.586,Z 441.69,A -85,B 0,C 180,E1 -8218.775,E2 -8218.775} C_VEL
LIN {X 0,Y 452.47,Z 443.661,A -85,B 0,C 180,E1 -8219.803,E2 -8219.803} C_VEL
LIN {X 0,Y 452.386,Z 445.584,A -85,B 0,C 180,E1 -8221.317,E2 -8221.317} C_VEL
LIN {X 0,Y 452.313,Z 446.382,A -85,B 0,C 180,E1 -8222.975,E2 -8222.975} C_VEL
LIN {X 0,Y 452.341,Z 445.823,A -85,B 0,C 180,E1 -8224.581,E2 -8224.581} C_VEL
LIN {X 0,Y 452.436,Z 443.966,A -85,B 0,C 180,E1 -8226.176,E2 -8226.176} C_VEL
LIN {X 0,Y 452.625,Z 441.072,A -85,B 0,C 180,E1 -8227.65,E2 -8227.65} C_VEL
LIN {X 0,Y 452.791,Z 437.011,A -85,B 0,C 180,E1 -8229.11,E2 -8229.11} C_VEL
LIN {X 0,Y 453.065,Z 431.275,A -85,B 0,C 180,E1 -8230.654,E2 -8230.654} C_VEL
LIN {X 0,Y 453.454,Z 424.061,A -85,B 0,C 180,E1 -8232.14,E2 -8232.14} C_VEL
LIN {X 0,Y 453.935,Z 416.207,A -85,B 0,C 180,E1 -8233.433,E2 -8233.433} C_VEL
LIN {X 0,Y 454.451,Z 406.992,A -85,B 0,C 180,E1 -8234.663,E2 -8234.663} C_VEL
LIN {X 0,Y 454.932,Z 397.932,A -85,B 0,C 180,E1 -8235.646,E2 -8235.646} C_VEL
LIN {X 0,Y 455.517,Z 386.578,A -85,B 0,C 180,E1 -8236.639,E2 -8236.639} C_VEL
LIN {X 0,Y 456.077,Z 374.81,A -85,B 0,C 180,E1 -8237.448,E2 -8237.448} C_VEL
LIN {X 0,Y 456.466,Z 363.124,A -85,B 0,C 180,E1 -8238.058,E2 -8238.058} C_VEL
LIN {X 0,Y 456.83,Z 349.781,A -85,B 0,C 180,E1 -8238.553,E2 -8238.553} C_VEL
LIN {X 0,Y 457.104,Z 336.502,A -85,B 0,C 180,E1 -8238.853,E2 -8238.853} C_VEL
LIN {X 0,Y 457.82,Z 251.12,A -85,B 0,C 180,E1 -8240.237,E2 -8240.237} C_VEL
LIN {X 0,Y 454.681,Z 235.577,A -85,B 0,C 180,E1 -8240.647,E2 -8240.647} C_VEL
LIN {X 0,Y 454.788,Z 225.054,A -85,B 0,C 180,E1 -8242.714,E2 -8242.714} C_VEL
LIN {X 0,Y 453.463,Z 218.001,A -85,B 0,C 180,E1 -8244.201,E2 -8244.201} C_VEL
LIN {X 0,Y 453.445,Z 218.006,A -85,B 0,C 180,E1 -8247.156,E2 -8247.156} C_VEL
LIN {X 0,Y 453.479,Z 217.997,A -85,B 0,C 180,E1 -8250.276,E2 -8250.276} C_VEL
LIN {X 0,Y 453.481,Z 217.998,A -85,B 0,C 180,E1 -8253.3,E2 -8253.3} C_VEL
LIN {X 0,Y 453.473,Z 217.996,A -85,B 0,C 180,E1 -8256.244,E2 -8256.244} C_VEL
LIN {X 0,Y 453.454,Z 218.004,A -85,B 0,C 180,E1 -8259.123,E2 -8259.123} C_VEL
LIN {X 0,Y 453.485,Z 217.995,A -85,B 0,C 180,E1 -8261.95,E2 -8261.95} C_VEL
LIN {X 0,Y 453.516,Z 217.997,A -85,B 0,C 180,E1 -8264.732,E2 -8264.732} C_VEL
LIN {X 0,Y 453.582,Z 217.982,A -85,B 0,C 180,E1 -8267.478,E2 -8267.478} C_VEL
LIN {X 0,Y 453.569,Z 217.985,A -85,B 0,C 180,E1 -8271.092,E2 -8271.092} C_VEL
LIN {X 0,Y 453.646,Z 217.973,A -85,B 0,C 180,E1 -8273.78,E2 -8273.78} C_VEL
LIN {X 0,Y 453.727,Z 217.963,A -85,B 0,C 180,E1 -8277.342,E2 -8277.342} C_VEL
LIN {X 0,Y 453.806,Z 217.953,A -85,B 0,C 180,E1 -8280.005,E2 -8280.005} C_VEL
LIN {X 0,Y 453.7,Z 217.968,A -85,B 0,C 180,E1 -8282.668,E2 -8282.668} C_VEL
LIN {X 0,Y 453.647,Z 217.971,A -85,B 0,C 180,E1 -8286.23,E2 -8286.23} C_VEL
LIN {X 0,Y 453.567,Z 217.984,A -85,B 0,C 180,E1 -8288.918,E2 -8288.918} C_VEL
LIN {X 0,Y 453.56,Z 217.99,A -85,B 0,C 180,E1 -8292.533,E2 -8292.533} C_VEL
LIN {X 0,Y 453.542,Z 217.988,A -85,B 0,C 180,E1 -8296.2,E2 -8296.2} C_VEL
LIN {X 0,Y 453.516,Z 217.991,A -85,B 0,C 180,E1 -8299.043,E2 -8299.043} C_VEL
LIN {X 0,Y 453.475,Z 217.994,A -85,B 0,C 180,E1 -8301.84,E2 -8301.84} C_VEL
LIN {X 0,Y 453.462,Z 218,A -85,B 0,C 180,E1 -8304.741,E2 -8304.741} C_VEL
LIN {X 0,Y 453.464,Z 217.996,A -85,B 0,C 180,E1 -8307.946,E2 -8307.946} C_VEL
LIN {X 0,Y 453.46,Z 218.001,A -85,B 0,C 180,E1 -8310.765,E2 -8310.765} C_VEL
LIN {X 0,Y 453.468,Z 217.994,A -85,B 0,C 180,E1 -8313.917,E2 -8313.917} C_VEL
LIN {X 0,Y 453.438,Z 217.999,A -85,B 0,C 180,E1 -8317.195,E2 -8317.195} C_VEL
LIN {X 0,Y 453.47,Z 218.002,A -85,B 0,C 180,E1 -8320.615,E2 -8320.615} C_VEL
LIN {X 0,Y 453.483,Z 218,A -85,B 0,C 180,E1 -8324.53,E2 -8324.53} C_VEL
LIN {X 0,Y 453.443,Z 218.007,A -85,B 0,C 180,E1 -8328.207,E2 -8328.207} C_VEL
LIN {X 0,Y 453.428,Z 218.003,A -85,B 0,C 180,E1 -8330.807,E2 -8330.807} C_VEL
LIN {X 0,Y 453.443,Z 218.004,A -85,B 0,C 180,E1 -8333.917,E2 -8333.917} C_VEL
LIN {X 0,Y 453.471,Z 218,A -85,B 0,C 180,E1 -8336.819,E2 -8336.819} C_VEL
LIN {X 0,Y 453.457,Z 218.006,A -85,B 0,C 180,E1 -8340.268,E2 -8340.268} C_VEL
LIN {X 0,Y 453.429,Z 218.005,A -85,B 0,C 180,E1 -8343.29,E2 -8343.29} C_VEL
LIN {X 0,Y 453.468,Z 218.11,A -85,B 0,C 180,E1 -8343.656,E2 -8343.656} C_VEL
LIN {X 0,Y 455.757,Z 229.941,A -85,B 0,C 180,E1 -8345.947,E2 -8345.947} C_VEL
LIN {X 0,Y 455.66,Z 236.242,A -85,B 0,C 180,E1 -8347.08,E2 -8347.08} C_VEL
LIN {X 0,Y 454.793,Z 255.65,A -85,B 0,C 180,E1 -8350.506,E2 -8350.506} C_VEL
LIN {X 0,Y 454.378,Z 266.701,A -85,B 0,C 180,E1 -8352.4,E2 -8352.4} C_VEL
LIN {X 0,Y 457.613,Z 288.173,A -85,B 0,C 180,E1 -8352.888,E2 -8352.888} C_VEL
LIN {X 0,Y 456.844,Z 375.669,A -85,B 0,C 180,E1 -8354.326,E2 -8354.326} C_VEL
LIN {X 0,Y 456.362,Z 389.442,A -85,B 0,C 180,E1 -8354.738,E2 -8354.738} C_VEL
LIN {X 0,Y 455.877,Z 401.304,A -85,B 0,C 180,E1 -8355.264,E2 -8355.264} C_VEL
LIN {X 0,Y 455.328,Z 412.556,A -85,B 0,C 180,E1 -8355.931,E2 -8355.931} C_VEL
LIN {X 0,Y 454.805,Z 423.86,A -85,B 0,C 180,E1 -8356.793,E2 -8356.793} C_VEL
LIN {X 0,Y 454.257,Z 434.74,A -85,B 0,C 180,E1 -8357.831,E2 -8357.831} C_VEL
LIN {X 0,Y 453.774,Z 443.345,A -85,B 0,C 180,E1 -8358.837,E2 -8358.837} C_VEL
LIN {X 0,Y 453.315,Z 451.287,A -85,B 0,C 180,E1 -8359.956,E2 -8359.956} C_VEL
LIN {X 0,Y 452.992,Z 459.051,A -85,B 0,C 180,E1 -8361.3,E2 -8361.3} C_VEL
LIN {X 0,Y 452.683,Z 466.206,A -85,B 0,C 180,E1 -8362.866,E2 -8362.866} C_VEL
LIN {X 0,Y 452.54,Z 470.972,A -85,B 0,C 180,E1 -8364.207,E2 -8364.207} C_VEL
LIN {X 0,Y 452.489,Z 474.617,A -85,B 0,C 180,E1 -8365.546,E2 -8365.546} C_VEL
LIN {X 0,Y 452.485,Z 476.498,A -85,B 0,C 180,E1 -8366.438,E2 -8366.438} C_VEL
LIN {X 0,Y 452.512,Z 477.911,A -85,B 0,C 180,E1 -8367.33,E2 -8367.33} C_VEL
LIN {X 0,Y 452.436,Z 479.535,A -85,B 0,C 180,E1 -8369.11,E2 -8369.11} C_VEL
LIN {X 0,Y 452.442,Z 479.754,A -85,B 0,C 180,E1 -8370,E2 -8370} C_VEL
LIN {X 0,Y 452.461,Z 478.925,A -85,B 0,C 180,E1 -8371.78,E2 -8371.78} C_VEL
LIN {X 0,Y 452.512,Z 477.924,A -85,B 0,C 180,E1 -8372.671,E2 -8372.671} C_VEL
LIN {X 0,Y 452.486,Z 476.508,A -85,B 0,C 180,E1 -8373.562,E2 -8373.562} C_VEL
LIN {X 0,Y 452.546,Z 473.545,A -85,B 0,C 180,E1 -8374.9,E2 -8374.9} C_VEL
LIN {X 0,Y 452.622,Z 468.973,A -85,B 0,C 180,E1 -8376.396,E2 -8376.396} C_VEL
LIN {X 0,Y 452.842,Z 462.321,A -85,B 0,C 180,E1 -8378.029,E2 -8378.029} C_VEL
LIN {X 0,Y 453.114,Z 455.335,A -85,B 0,C 180,E1 -8379.373,E2 -8379.373} C_VEL
LIN {X 0,Y 453.513,Z 446.574,A -85,B 0,C 180,E1 -8380.717,E2 -8380.717} C_VEL
LIN {X 0,Y 454.069,Z 437.607,A -85,B 0,C 180,E1 -8381.834,E2 -8381.834} C_VEL
LIN {X 0,Y 454.617,Z 426.61,A -85,B 0,C 180,E1 -8382.946,E2 -8382.946} C_VEL
LIN {X 0,Y 455.156,Z 415.302,A -85,B 0,C 180,E1 -8383.847,E2 -8383.847} C_VEL
LIN {X 0,Y 455.706,Z 402.714,A -85,B 0,C 180,E1 -8384.627,E2 -8384.627} C_VEL
LIN {X 0,Y 456.267,Z 389.792,A -85,B 0,C 180,E1 -8385.208,E2 -8385.208} C_VEL
LIN {X 0,Y 456.634,Z 377.132,A -85,B 0,C 180,E1 -8385.596,E2 -8385.596} C_VEL
LIN {X 0,Y 457.023,Z 348.167,A -85,B 0,C 180,E1 -8386.09,E2 -8386.09} C_VEL
LIN {X 0,Y 457.413,Z 287.136,A -85,B 0,C 180,E1 -8387.077,E2 -8387.077} C_VEL
LIN {X 0,Y 454.348,Z 267.101,A -85,B 0,C 180,E1 -8387.527,E2 -8387.527} C_VEL
LIN {X 0,Y 455.19,Z 248.699,A -85,B 0,C 180,E1 -8390.8,E2 -8390.8} C_VEL
LIN {X 0,Y 455.971,Z 233.046,A -85,B 0,C 180,E1 -8393.624,E2 -8393.624} C_VEL
LIN {X 0,Y 455.601,Z 228.547,A -85,B 0,C 180,E1 -8394.474,E2 -8394.474} C_VEL
LIN {X 0,Y 453.47,Z 218.001,A -85,B 0,C 180,E1 -8396.572,E2 -8396.572} C_VEL
LIN {X 0,Y 453.46,Z 218.003,A -85,B 0,C 180,E1 -8399.778,E2 -8399.778} C_VEL
LIN {X 0,Y 453.454,Z 217.997,A -85,B 0,C 180,E1 -8403.178,E2 -8403.178} C_VEL
LIN {X 0,Y 453.416,Z 218.003,A -85,B 0,C 180,E1 -8406.289,E2 -8406.289} C_VEL
LIN {X 0,Y 453.425,Z 218.004,A -85,B 0,C 180,E1 -8409.455,E2 -8409.455} C_VEL
LIN {X 0,Y 453.436,Z 218.004,A -85,B 0,C 180,E1 -8411.925,E2 -8411.925} C_VEL
LIN {X 0,Y 453.462,Z 218,A -85,B 0,C 180,E1 -8415.473,E2 -8415.473} C_VEL
LIN {X 0,Y 453.442,Z 218,A -85,B 0,C 180,E1 -8418.201,E2 -8418.201} C_VEL
LIN {X 0,Y 453.425,Z 218,A -85,B 0,C 180,E1 -8420.802,E2 -8420.802} C_VEL
LIN {X 0,Y 453.408,Z 218.007,A -85,B 0,C 180,E1 -8423.909,E2 -8423.909} C_VEL
LIN {X 0,Y 453.455,Z 217.998,A -85,B 0,C 180,E1 -8427.145,E2 -8427.145} C_VEL
LIN {X 0,Y 453.451,Z 217.998,A -85,B 0,C 180,E1 -8430.263,E2 -8430.263} C_VEL
LIN {X 0,Y 453.415,Z 218.004,A -85,B 0,C 180,E1 -8433.284,E2 -8433.284} C_VEL
LIN {X 0,Y 453.491,Z 217.993,A -85,B 0,C 180,E1 -8436.234,E2 -8436.234} C_VEL
LIN {X 0,Y 453.464,Z 217.997,A -85,B 0,C 180,E1 -8439.113,E2 -8439.113} C_VEL
LIN {X 0,Y 453.465,Z 217.999,A -85,B 0,C 180,E1 -8441.938,E2 -8441.938} C_VEL
LIN {X 0,Y 453.525,Z 217.987,A -85,B 0,C 180,E1 -8444.722,E2 -8444.722} C_VEL
LIN {X 0,Y 453.561,Z 217.99,A -85,B 0,C 180,E1 -8447.467,E2 -8447.467} C_VEL
LIN {X 0,Y 453.547,Z 217.987,A -85,B 0,C 180,E1 -8451.081,E2 -8451.081} C_VEL
LIN {X 0,Y 453.626,Z 217.98,A -85,B 0,C 180,E1 -8453.769,E2 -8453.769} C_VEL
LIN {X 0,Y 453.673,Z 217.974,A -85,B 0,C 180,E1 -8457.331,E2 -8457.331} C_VEL
LIN {X 0,Y 453.732,Z 217.964,A -85,B 0,C 180,E1 -8459.995,E2 -8459.995} C_VEL
LIN {X 0,Y 453.698,Z 217.966,A -85,B 0,C 180,E1 -8462.658,E2 -8462.658} C_VEL
LIN {X 0,Y 453.61,Z 217.977,A -85,B 0,C 180,E1 -8466.221,E2 -8466.221} C_VEL
LIN {X 0,Y 453.542,Z 217.987,A -85,B 0,C 180,E1 -8468.909,E2 -8468.909} C_VEL
LIN {X 0,Y 453.544,Z 217.985,A -85,B 0,C 180,E1 -8472.523,E2 -8472.523} C_VEL
LIN {X 0,Y 453.521,Z 217.988,A -85,B 0,C 180,E1 -8476.191,E2 -8476.191} C_VEL
LIN {X 0,Y 453.491,Z 217.995,A -85,B 0,C 180,E1 -8479.034,E2 -8479.034} C_VEL
LIN {X 0,Y 453.447,Z 218,A -85,B 0,C 180,E1 -8481.831,E2 -8481.831} C_VEL
LIN {X 0,Y 453.46,Z 217.996,A -85,B 0,C 180,E1 -8484.73,E2 -8484.73} C_VEL
LIN {X 0,Y 453.495,Z 217.992,A -85,B 0,C 180,E1 -8487.953,E2 -8487.953} C_VEL
LIN {X 0,Y 453.428,Z 218.005,A -85,B 0,C 180,E1 -8491.52,E2 -8491.52} C_VEL
LIN {X 0,Y 453.447,Z 217.999,A -85,B 0,C 180,E1 -8494.772,E2 -8494.772} C_VEL
LIN {X 0,Y 453.421,Z 218,A -85,B 0,C 180,E1 -8498.307,E2 -8498.307} C_VEL
LIN {X 0,Y 453.45,Z 217.997,A -85,B 0,C 180,E1 -8500.604,E2 -8500.604} C_VEL
LIN {X 0,Y 453.424,Z 218,A -85,B 0,C 180,E1 -8504.216,E2 -8504.216} C_VEL
LIN {X 0,Y 453.414,Z 218.006,A -85,B 0,C 180,E1 -8507.001,E2 -8507.001} C_VEL
LIN {X 0,Y 453.444,Z 218.003,A -85,B 0,C 180,E1 -8509.405,E2 -8509.405} C_VEL
LIN {X 0,Y 453.421,Z 218,A -85,B 0,C 180,E1 -8512.219,E2 -8512.219} C_VEL
LIN {X 0,Y 453.435,Z 218.007,A -85,B 0,C 180,E1 -8515.219,E2 -8515.219} C_VEL
LIN {X 0,Y 453.411,Z 218.002,A -85,B 0,C 180,E1 -8518.471,E2 -8518.471} C_VEL
LIN {X 0,Y 453.457,Z 218.003,A -85,B 0,C 180,E1 -8521.285,E2 -8521.285} C_VEL
LIN {X 0,Y 453.482,Z 217.993,A -85,B 0,C 180,E1 -8524.283,E2 -8524.283} C_VEL
LIN {X 0,Y 453.44,Z 218.006,A -85,B 0,C 180,E1 -8527.203,E2 -8527.203} C_VEL
LIN {X 0,Y 453.451,Z 217.997,A -85,B 0,C 180,E1 -8530.064,E2 -8530.064} C_VEL
LIN {X 0,Y 453.453,Z 218.001,A -85,B 0,C 180,E1 -8532.874,E2 -8532.874} C_VEL
LIN {X 0,Y 453.454,Z 217.998,A -85,B 0,C 180,E1 -8535.642,E2 -8535.642} C_VEL
LIN {X 0,Y 453.526,Z 217.988,A -85,B 0,C 180,E1 -8538.378,E2 -8538.378} C_VEL
LIN {X 0,Y 453.593,Z 217.979,A -85,B 0,C 180,E1 -8541.984,E2 -8541.984} C_VEL
LIN {X 0,Y 453.587,Z 217.983,A -85,B 0,C 180,E1 -8543.04,E2 -8543.04} C_VEL
LIN {X 0,Y 452.901,Z 218.067,A -85,B 0,C 180,E1 -8543.781,E2 -8543.781} C_VEL
LIN {X 0,Y 449.953,Z 218.439,A -85,B 0,C 180,E1 -8544.983,E2 -8544.983} C_VEL
LIN {X 0,Y 447.528,Z 218.737,A -85,B 0,C 180,E1 -8545.952,E2 -8545.952} C_VEL
LIN {X 0,Y 446.583,Z 218.856,A -85,B 0,C 180,E1 -8546.703,E2 -8546.703} C_VEL
LIN {X 0,Y 446.558,Z 218.857,A -85,B 0,C 180,E1 -8546.956,E2 -8546.956} C_VEL
LIN {X 0,Y 446.728,Z 218.834,A -85,B 0,C 180,E1 -8550,E2 -8550} C_VEL
LIN {X 0,Y 446.653,Z 218.847,A -85,B 0,C 180,E1 -8552.705,E2 -8552.705} C_VEL
LIN {X 0,Y 446.599,Z 218.851,A -85,B 0,C 180,E1 -8556.324,E2 -8556.324} C_VEL
LIN {X 0,Y 446.497,Z 218.87,A -85,B 0,C 180,E1 -8559.056,E2 -8559.056} C_VEL
LIN {X 0,Y 446.533,Z 219.025,A -85,B 0,C 180,E1 -8561.576,E2 -8561.576} C_VEL
LIN {X 0,Y 447.84,Z 227.035,A -85,B 0,C 180,E1 -8563.388,E2 -8563.388} C_VEL
LIN {X 0,Y 447.604,Z 235.857,A -85,B 0,C 180,E1 -8565.277,E2 -8565.277} C_VEL
LIN {X 0,Y 450.962,Z 253.477,A -85,B 0,C 180,E1 -8565.71,E2 -8565.71} C_VEL
LIN {X 0,Y 449.958,Z 343.631,A -85,B 0,C 180,E1 -8567.204,E2 -8567.204} C_VEL
LIN {X 0,Y 449.606,Z 357.104,A -85,B 0,C 180,E1 -8567.618,E2 -8567.618} C_VEL
LIN {X 0,Y 449.269,Z 368.603,A -85,B 0,C 180,E1 -8568.138,E2 -8568.138} C_VEL
LIN {X 0,Y 448.828,Z 380.273,A -85,B 0,C 180,E1 -8568.841,E2 -8568.841} C_VEL
LIN {X 0,Y 448.251,Z 391.61,A -85,B 0,C 180,E1 -8569.723,E2 -8569.723} C_VEL
LIN {X 0,Y 447.715,Z 401.513,A -85,B 0,C 180,E1 -8570.682,E2 -8570.682} C_VEL
LIN {X 0,Y 447.122,Z 411.519,A -85,B 0,C 180,E1 -8571.876,E2 -8571.876} C_VEL
LIN {X 0,Y 446.636,Z 420.156,A -85,B 0,C 180,E1 -8573.165,E2 -8573.165} C_VEL
LIN {X 0,Y 446.238,Z 427.017,A -85,B 0,C 180,E1 -8574.419,E2 -8574.419} C_VEL
LIN {X 0,Y 445.935,Z 432.385,A -85,B 0,C 180,E1 -8575.617,E2 -8575.617} C_VEL
LIN {X 0,Y 445.672,Z 438.022,A -85,B 0,C 180,E1 -8577.213,E2 -8577.213} C_VEL
LIN {X 0,Y 445.516,Z 442.043,A -85,B 0,C 180,E1 -8578.759,E2 -8578.759} C_VEL
LIN {X 0,Y 445.348,Z 444.781,A -85,B 0,C 180,E1 -8580.33,E2 -8580.33} C_VEL
LIN {X 0,Y 445.274,Z 446.074,A -85,B 0,C 180,E1 -8581.551,E2 -8581.551} C_VEL
LIN {X 0,Y 445.236,Z 446.633,A -85,B 0,C 180,E1 -8583.232,E2 -8583.232} C_VEL
LIN {X 0,Y 445.261,Z 445.878,A -85,B 0,C 180,E1 -8584.852,E2 -8584.852} C_VEL
LIN {X 0,Y 445.365,Z 443.928,A -85,B 0,C 180,E1 -8586.423,E2 -8586.423} C_VEL
LIN {X 0,Y 445.567,Z 440.8,A -85,B 0,C 180,E1 -8587.962,E2 -8587.962} C_VEL
LIN {X 0,Y 445.786,Z 436.586,A -85,B 0,C 180,E1 -8589.433,E2 -8589.433} C_VEL
LIN {X 0,Y 446.036,Z 431.153,A -85,B 0,C 180,E1 -8590.871,E2 -8590.871} C_VEL
LIN {X 0,Y 446.455,Z 424.327,A -85,B 0,C 180,E1 -8592.292,E2 -8592.292} C_VEL
LIN {X 0,Y 446.851,Z 417.572,A -85,B 0,C 180,E1 -8593.438,E2 -8593.438} C_VEL
LIN {X 0,Y 447.411,Z 408.792,A -85,B 0,C 180,E1 -8594.662,E2 -8594.662} C_VEL
LIN {X 0,Y 447.942,Z 399.586,A -85,B 0,C 180,E1 -8595.712,E2 -8595.712} C_VEL
LIN {X 0,Y 448.539,Z 388.711,A -85,B 0,C 180,E1 -8596.71,E2 -8596.71} C_VEL
LIN {X 0,Y 449.116,Z 377.11,A -85,B 0,C 180,E1 -8597.55,E2 -8597.55} C_VEL
LIN {X 0,Y 449.605,Z 364.975,A -85,B 0,C 180,E1 -8598.226,E2 -8598.226} C_VEL
LIN {X 0,Y 449.96,Z 352.062,A -85,B 0,C 180,E1 -8598.739,E2 -8598.739} C_VEL
LIN {X 0,Y 450.253,Z 338.642,A -85,B 0,C 180,E1 -8599.073,E2 -8599.073} C_VEL
LIN {X 0,Y 451.14,Z 252.288,A -85,B 0,C 180,E1 -8600.496,E2 -8600.496} C_VEL
LIN {X 0,Y 447.786,Z 235.819,A -85,B 0,C 180,E1 -8600.941,E2 -8600.941} C_VEL
LIN {X 0,Y 447.858,Z 226.304,A -85,B 0,C 180,E1 -8602.838,E2 -8602.838} C_VEL
LIN {X 0,Y 446.429,Z 218.878,A -85,B 0,C 180,E1 -8604.428,E2 -8604.428} C_VEL
LIN {X 0,Y 446.385,Z 218.883,A -85,B 0,C 180,E1 -8607.644,E2 -8607.644} C_VEL
LIN {X 0,Y 446.435,Z 218.878,A -85,B 0,C 180,E1 -8610.797,E2 -8610.797} C_VEL
LIN {X 0,Y 446.446,Z 218.87,A -85,B 0,C 180,E1 -8613.854,E2 -8613.854} C_VEL
LIN {X 0,Y 446.399,Z 218.883,A -85,B 0,C 180,E1 -8616.829,E2 -8616.829} C_VEL
LIN {X 0,Y 446.416,Z 218.875,A -85,B 0,C 180,E1 -8619.743,E2 -8619.743} C_VEL
LIN {X 0,Y 446.438,Z 218.877,A -85,B 0,C 180,E1 -8622.603,E2 -8622.603} C_VEL
LIN {X 0,Y 446.446,Z 218.872,A -85,B 0,C 180,E1 -8625.418,E2 -8625.418} C_VEL
LIN {X 0,Y 446.52,Z 218.861,A -85,B 0,C 180,E1 -8628.199,E2 -8628.199} C_VEL
LIN {X 0,Y 446.516,Z 218.864,A -85,B 0,C 180,E1 -8630.95,E2 -8630.95} C_VEL
LIN {X 0,Y 446.615,Z 218.849,A -85,B 0,C 180,E1 -8633.681,E2 -8633.681} C_VEL
LIN {X 0,Y 446.674,Z 218.842,A -85,B 0,C 180,E1 -8637.3,E2 -8637.3} C_VEL
LIN {X 0,Y 446.776,Z 218.829,A -85,B 0,C 180,E1 -8640.005,E2 -8640.005} C_VEL
LIN {X 0,Y 446.65,Z 218.847,A -85,B 0,C 180,E1 -8642.711,E2 -8642.711} C_VEL
LIN {X 0,Y 446.617,Z 218.848,A -85,B 0,C 180,E1 -8646.329,E2 -8646.329} C_VEL
LIN {X 0,Y 446.515,Z 218.861,A -85,B 0,C 180,E1 -8649.06,E2 -8649.06} C_VEL
LIN {X 0,Y 446.518,Z 218.866,A -85,B 0,C 180,E1 -8652.734,E2 -8652.734} C_VEL
LIN {X 0,Y 446.486,Z 218.871,A -85,B 0,C 180,E1 -8656.463,E2 -8656.463} C_VEL
LIN {X 0,Y 446.467,Z 218.867,A -85,B 0,C 180,E1 -8659.307,E2 -8659.307} C_VEL
LIN {X 0,Y 446.416,Z 218.876,A -85,B 0,C 180,E1 -8662.204,E2 -8662.204} C_VEL
LIN {X 0,Y 446.413,Z 218.874,A -85,B 0,C 180,E1 -8665.159,E2 -8665.159} C_VEL
LIN {X 0,Y 446.439,Z 218.873,A -85,B 0,C 180,E1 -8668.186,E2 -8668.186} C_VEL
LIN {X 0,Y 446.411,Z 218.875,A -85,B 0,C 180,E1 -8671.305,E2 -8671.305} C_VEL
LIN {X 0,Y 446.423,Z 218.878,A -85,B 0,C 180,E1 -8674.527,E2 -8674.527} C_VEL
LIN {X 0,Y 446.398,Z 218.879,A -85,B 0,C 180,E1 -8678.078,E2 -8678.078} C_VEL
LIN {X 0,Y 446.401,Z 218.878,A -85,B 0,C 180,E1 -8681.398,E2 -8681.398} C_VEL
LIN {X 0,Y 446.419,Z 218.877,A -85,B 0,C 180,E1 -8685.112,E2 -8685.112} C_VEL
LIN {X 0,Y 446.402,Z 218.881,A -85,B 0,C 180,E1 -8688.607,E2 -8688.607} C_VEL
LIN {X 0,Y 446.392,Z 218.884,A -85,B 0,C 180,E1 -8692.121,E2 -8692.121} C_VEL
LIN {X 0,Y 446.418,Z 218.876,A -85,B 0,C 180,E1 -8695.477,E2 -8695.477} C_VEL
LIN {X 0,Y 446.397,Z 218.883,A -85,B 0,C 180,E1 -8698.699,E2 -8698.699} C_VEL
LIN {X 0,Y 446.406,Z 218.882,A -85,B 0,C 180,E1 -8701.845,E2 -8701.845} C_VEL
LIN {X 0,Y 446.4,Z 218.966,A -85,B 0,C 180,E1 -8703.411,E2 -8703.411} C_VEL
LIN {X 0,Y 448.751,Z 230.861,A -85,B 0,C 180,E1 -8705.759,E2 -8705.759} C_VEL
LIN {X 0,Y 448.875,Z 234.689,A -85,B 0,C 180,E1 -8706.469,E2 -8706.469} C_VEL
LIN {X 0,Y 448.05,Z 250.639,A -85,B 0,C 180,E1 -8709.334,E2 -8709.334} C_VEL
LIN {X 0,Y 447.408,Z 266.305,A -85,B 0,C 180,E1 -8712.102,E2 -8712.102} C_VEL
LIN {X 0,Y 450.843,Z 289.307,A -85,B 0,C 180,E1 -8712.638,E2 -8712.638} C_VEL
LIN {X 0,Y 450.022,Z 375.687,A -85,B 0,C 180,E1 -8714.082,E2 -8714.082} C_VEL
LIN {X 0,Y 449.523,Z 389.358,A -85,B 0,C 180,E1 -8714.5,E2 -8714.5} C_VEL
LIN {X 0,Y 448.963,Z 402.209,A -85,B 0,C 180,E1 -8715.09,E2 -8715.09} C_VEL
LIN {X 0,Y 448.341,Z 413.967,A -85,B 0,C 180,E1 -8715.823,E2 -8715.823} C_VEL
LIN {X 0,Y 447.758,Z 425.761,A -85,B 0,C 180,E1 -8716.768,E2 -8716.768} C_VEL
LIN {X 0,Y 447.233,Z 435.585,A -85,B 0,C 180,E1 -8717.752,E2 -8717.752} C_VEL
LIN {X 0,Y 446.657,Z 444.813,A -85,B 0,C 180,E1 -8718.887,E2 -8718.887} C_VEL
LIN {X 0,Y 446.156,Z 453.811,A -85,B 0,C 180,E1 -8720.251,E2 -8720.251} C_VEL
LIN {X 0,Y 445.819,Z 461.06,A -85,B 0,C 180,E1 -8721.616,E2 -8721.616} C_VEL
LIN {X 0,Y 445.612,Z 465.958,A -85,B 0,C 180,E1 -8722.752,E2 -8722.752} C_VEL
LIN {X 0,Y 445.465,Z 470.276,A -85,B 0,C 180,E1 -8723.974,E2 -8723.974} C_VEL
LIN {X 0,Y 445.415,Z 474.365,A -85,B 0,C 180,E1 -8725.475,E2 -8725.475} C_VEL
LIN {X 0,Y 445.384,Z 476.243,A -85,B 0,C 180,E1 -8726.381,E2 -8726.381} C_VEL
LIN {X 0,Y 445.438,Z 477.655,A -85,B 0,C 180,E1 -8727.287,E2 -8727.287} C_VEL
LIN {X 0,Y 445.346,Z 479.276,A -85,B 0,C 180,E1 -8729.096,E2 -8729.096} C_VEL
LIN {X 0,Y 445.35,Z 479.491,A -85,B 0,C 180,E1 -8730,E2 -8730} C_VEL
LIN {X 0,Y 445.379,Z 478.657,A -85,B 0,C 180,E1 -8731.809,E2 -8731.809} C_VEL
LIN {X 0,Y 445.438,Z 477.654,A -85,B 0,C 180,E1 -8732.713,E2 -8732.713} C_VEL
LIN {X 0,Y 445.385,Z 476.232,A -85,B 0,C 180,E1 -8733.619,E2 -8733.619} C_VEL
LIN {X 0,Y 445.474,Z 473.263,A -85,B 0,C 180,E1 -8734.978,E2 -8734.978} C_VEL
LIN {X 0,Y 445.541,Z 469.081,A -85,B 0,C 180,E1 -8736.385,E2 -8736.385} C_VEL
LIN {X 0,Y 445.723,Z 463.034,A -85,B 0,C 180,E1 -8737.93,E2 -8737.93} C_VEL
LIN {X 0,Y 446.023,Z 456.269,A -85,B 0,C 180,E1 -8739.294,E2 -8739.294} C_VEL
LIN {X 0,Y 446.428,Z 447.871,A -85,B 0,C 180,E1 -8740.66,E2 -8740.66} C_VEL
LIN {X 0,Y 446.981,Z 439.222,A -85,B 0,C 180,E1 -8741.794,E2 -8741.794} C_VEL
LIN {X 0,Y 447.505,Z 429.056,A -85,B 0,C 180,E1 -8742.883,E2 -8742.883} C_VEL
LIN {X 0,Y 448.094,Z 417.978,A -85,B 0,C 180,E1 -8743.838,E2 -8743.838} C_VEL
LIN {X 0,Y 448.651,Z 406.241,A -85,B 0,C 180,E1 -8744.631,E2 -8744.631} C_VEL
LIN {X 0,Y 449.197,Z 394.057,A -85,B 0,C 180,E1 -8745.25,E2 -8745.25} C_VEL
LIN {X 0,Y 449.671,Z 380.794,A -85,B 0,C 180,E1 -8745.728,E2 -8745.728} C_VEL
LIN {X 0,Y 449.957,Z 367.794,A -85,B 0,C 180,E1 -8746.008,E2 -8746.008} C_VEL
LIN {X 0,Y 450.618,Z 288.025,A -85,B 0,C 180,E1 -8747.313,E2 -8747.313} C_VEL
LIN {X 0,Y 447.379,Z 266.805,A -85,B 0,C 180,E1 -8747.806,E2 -8747.806} C_VEL
LIN {X 0,Y 448.3,Z 248.405,A -85,B 0,C 180,E1 -8751.135,E2 -8751.135} C_VEL
LIN {X 0,Y 449.065,Z 232.742,A -85,B 0,C 180,E1 -8754.01,E2 -8754.01} C_VEL
LIN {X 0,Y 447.091,Z 222.171,A -85,B 0,C 180,E1 -8756.112,E2 -8756.112} C_VEL
LIN {X 0,Y 446.433,Z 218.877,A -85,B 0,C 180,E1 -8756.796,E2 -8756.796} C_VEL
LIN {X 0,Y 446.415,Z 218.878,A -85,B 0,C 180,E1 -8760.25,E2 -8760.25} C_VEL
LIN {X 0,Y 446.408,Z 218.877,A -85,B 0,C 180,E1 -8763.442,E2 -8763.442} C_VEL
LIN {X 0,Y 446.386,Z 218.877,A -85,B 0,C 180,E1 -8766.746,E2 -8766.746} C_VEL
LIN {X 0,Y 446.394,Z 218.878,A -85,B 0,C 180,E1 -8770.202,E2 -8770.202} C_VEL
LIN {X 0,Y 446.352,Z 218.887,A -85,B 0,C 180,E1 -8773.586,E2 -8773.586} C_VEL
LIN {X 0,Y 446.377,Z 218.879,A -85,B 0,C 180,E1 -8776.405,E2 -8776.405} C_VEL
LIN {X 0,Y 446.392,Z 218.883,A -85,B 0,C 180,E1 -8779.793,E2 -8779.793} C_VEL
LIN {X 0,Y 446.382,Z 218.88,A -85,B 0,C 180,E1 -8783.249,E2 -8783.249} C_VEL
LIN {X 0,Y 446.414,Z 218.873,A -85,B 0,C 180,E1 -8786.56,E2 -8786.56} C_VEL
LIN {X 0,Y 446.417,Z 218.877,A -85,B 0,C 180,E1 -8789.98,E2 -8789.98} C_VEL
LIN {X 0,Y 446.377,Z 218.878,A -85,B 0,C 180,E1 -8792.829,E2 -8792.829} C_VEL
LIN {X 0,Y 446.423,Z 218.876,A -85,B 0,C 180,E1 -8795.932,E2 -8795.932} C_VEL
LIN {X 0,Y 446.444,Z 218.87,A -85,B 0,C 180,E1 -8798.768,E2 -8798.768} C_VEL
LIN {X 0,Y 446.415,Z 218.881,A -85,B 0,C 180,E1 -8801.643,E2 -8801.643} C_VEL
LIN {X 0,Y 446.473,Z 218.866,A -85,B 0,C 180,E1 -8804.474,E2 -8804.474} C_VEL
LIN {X 0,Y 446.512,Z 218.866,A -85,B 0,C 180,E1 -8807.38,E2 -8807.38} C_VEL
LIN {X 0,Y 446.498,Z 218.864,A -85,B 0,C 180,E1 -8810.939,E2 -8810.939} C_VEL
LIN {X 0,Y 446.596,Z 218.857,A -85,B 0,C 180,E1 -8813.671,E2 -8813.671} C_VEL
LIN {X 0,Y 446.625,Z 218.852,A -85,B 0,C 180,E1 -8817.289,E2 -8817.289} C_VEL
LIN {X 0,Y 446.683,Z 218.842,A -85,B 0,C 180,E1 -8819.995,E2 -8819.995} C_VEL
LIN {X 0,Y 446.647,Z 218.844,A -85,B 0,C 180,E1 -8822.7,E2 -8822.7} C_VEL
LIN {X 0,Y 446.581,Z 218.853,A -85,B 0,C 180,E1 -8826.319,E2 -8826.319} C_VEL
LIN {X 0,Y 446.493,Z 218.866,A -85,B 0,C 180,E1 -8829.051,E2 -8829.051} C_VEL
LIN {X 0,Y 446.501,Z 218.863,A -85,B 0,C 180,E1 -8832.724,E2 -8832.724} C_VEL
LIN {X 0,Y 446.464,Z 218.867,A -85,B 0,C 180,E1 -8836.454,E2 -8836.454} C_VEL
LIN {X 0,Y 446.442,Z 218.876,A -85,B 0,C 180,E1 -8839.298,E2 -8839.298} C_VEL
LIN {X 0,Y 446.387,Z 218.877,A -85,B 0,C 180,E1 -8842.194,E2 -8842.194} C_VEL
LIN {X 0,Y 446.405,Z 218.879,A -85,B 0,C 180,E1 -8845.148,E2 -8845.148} C_VEL
LIN {X 0,Y 446.452,Z 218.869,A -85,B 0,C 180,E1 -8848.173,E2 -8848.173} C_VEL
LIN {X 0,Y 446.381,Z 218.88,A -85,B 0,C 180,E1 -8851.769,E2 -8851.769} C_VEL
LIN {X 0,Y 446.389,Z 218.877,A -85,B 0,C 180,E1 -8854.518,E2 -8854.518} C_VEL
LIN {X 0,Y 446.372,Z 218.879,A -85,B 0,C 180,E1 -8858.074,E2 -8858.074} C_VEL
LIN {X 0,Y 446.383,Z 218.88,A -85,B 0,C 180,E1 -8860.913,E2 -8860.913} C_VEL
LIN {X 0,Y 446.375,Z 218.88,A -85,B 0,C 180,E1 -8863.839,E2 -8863.839} C_VEL
LIN {X 0,Y 446.35,Z 218.881,A -85,B 0,C 180,E1 -8866.399,E2 -8866.399} C_VEL
LIN {X 0,Y 446.377,Z 218.883,A -85,B 0,C 180,E1 -8869.078,E2 -8869.078} C_VEL
LIN {X 0,Y 446.376,Z 218.878,A -85,B 0,C 180,E1 -8872.119,E2 -8872.119} C_VEL
LIN {X 0,Y 446.376,Z 218.882,A -85,B 0,C 180,E1 -8875.473,E2 -8875.473} C_VEL
LIN {X 0,Y 446.362,Z 218.882,A -85,B 0,C 180,E1 -8878.696,E2 -8878.696} C_VEL
LIN {X 0,Y 446.427,Z 218.873,A -85,B 0,C 180,E1 -8881.818,E2 -8881.818} C_VEL
LIN {X 0,Y 446.414,Z 218.877,A -85,B 0,C 180,E1 -8884.846,E2 -8884.846} C_VEL
LIN {X 0,Y 446.425,Z 218.872,A -85,B 0,C 180,E1 -8888.231,E2 -8888.231} C_VEL
LIN {X 0,Y 446.402,Z 218.877,A -85,B 0,C 180,E1 -8891.647,E2 -8891.647} C_VEL
LIN {X 0,Y 446.453,Z 218.869,A -85,B 0,C 180,E1 -8894.478,E2 -8894.478} C_VEL
LIN {X 0,Y 446.484,Z 218.864,A -85,B 0,C 180,E1 -8898.192,E2 -8898.192} C_VEL
LIN {X 0,Y 446.542,Z 218.858,A -85,B 0,C 180,E1 -8901.857,E2 -8901.857} C_VEL
LIN {X 0,Y 446.592,Z 218.853,A -85,B 0,C 180,E1 -8904.582,E2 -8904.582} C_VEL
LIN {X 0,Y 446.558,Z 218.857,A -85,B 0,C 180,E1 -8906.956,E2 -8906.956} C_VEL
LIN {X 0,Y 446.04,Z 218.927,A -85,B 0,C 180,E1 -8907.709,E2 -8907.709} C_VEL
LIN {X 0,Y 443.253,Z 219.282,A -85,B 0,C 180,E1 -8908.933,E2 -8908.933} C_VEL
LIN {X 0,Y 440.788,Z 219.589,A -85,B 0,C 180,E1 -8909.921,E2 -8909.921} C_VEL
LIN {X 0,Y 439.694,Z 219.719,A -85,B 0,C 180,E1 -8910.684,E2 -8910.684} C_VEL
LIN {X 0,Y 439.591,Z 219.729,A -85,B 0,C 180,E1 -8910.942,E2 -8910.942} C_VEL
LIN {X 0,Y 439.6,Z 219.726,A -85,B 0,C 180,E1 -8912.749,E2 -8912.749} C_VEL
LIN {X 0,Y 439.569,Z 219.727,A -85,B 0,C 180,E1 -8916.426,E2 -8916.426} C_VEL
LIN {X 0,Y 439.454,Z 219.747,A -85,B 0,C 180,E1 -8919.202,E2 -8919.202} C_VEL
LIN {X 0,Y 439.454,Z 219.779,A -85,B 0,C 180,E1 -8921.356,E2 -8921.356} C_VEL
LIN {X 0,Y 440.866,Z 228.152,A -85,B 0,C 180,E1 -8923.278,E2 -8923.278} C_VEL
LIN {X 0,Y 440.682,Z 236.059,A -85,B 0,C 180,E1 -8924.99,E2 -8924.99} C_VEL
LIN {X 0,Y 444.165,Z 254.178,A -85,B 0,C 180,E1 -8925.457,E2 -8925.457} C_VEL
LIN {X 0,Y 443.128,Z 342.898,A -85,B 0,C 180,E1 -8926.943,E2 -8926.943} C_VEL
LIN {X 0,Y 442.784,Z 356.162,A -85,B 0,C 180,E1 -8927.343,E2 -8927.343} C_VEL
LIN {X 0,Y 442.374,Z 369.23,A -85,B 0,C 180,E1 -8927.935,E2 -8927.935} C_VEL
LIN {X 0,Y 441.897,Z 381.035,A -85,B 0,C 180,E1 -8928.667,E2 -8928.667} C_VEL
LIN {X 0,Y 441.328,Z 391.987,A -85,B 0,C 180,E1 -8929.537,E2 -8929.537} C_VEL
LIN {X 0,Y 440.75,Z 402.108,A -85,B 0,C 180,E1 -8930.536,E2 -8930.536} C_VEL
LIN {X 0,Y 440.148,Z 411.576,A -85,B 0,C 180,E1 -8931.684,E2 -8931.684} C_VEL
LIN {X 0,Y 439.61,Z 420.638,A -85,B 0,C 180,E1 -8933.058,E2 -8933.058} C_VEL
LIN {X 0,Y 439.223,Z 426.959,A -85,B 0,C 180,E1 -8934.229,E2 -8934.229} C_VEL
LIN {X 0,Y 438.862,Z 433.064,A -85,B 0,C 180,E1 -8935.618,E2 -8935.618} C_VEL
LIN {X 0,Y 438.593,Z 438.408,A -85,B 0,C 180,E1 -8937.172,E2 -8937.172} C_VEL
LIN {X 0,Y 438.445,Z 442.386,A -85,B 0,C 180,E1 -8938.742,E2 -8938.742} C_VEL
LIN {X 0,Y 438.284,Z 444.676,A -85,B 0,C 180,E1 -8940.03,E2 -8940.03} C_VEL
LIN {X 0,Y 438.223,Z 445.747,A -85,B 0,C 180,E1 -8940.876,E2 -8940.876} C_VEL
LIN {X 0,Y 438.16,Z 446.581,A -85,B 0,C 180,E1 -8941.958,E2 -8941.958} C_VEL
LIN {X 0,Y 438.162,Z 446.854,A -85,B 0,C 180,E1 -8943.496,E2 -8943.496} C_VEL
LIN {X 0,Y 438.215,Z 445.82,A -85,B 0,C 180,E1 -8945.264,E2 -8945.264} C_VEL
LIN {X 0,Y 438.333,Z 443.821,A -85,B 0,C 180,E1 -8946.723,E2 -8946.723} C_VEL
LIN {X 0,Y 438.525,Z 440.541,A -85,B 0,C 180,E1 -8948.265,E2 -8948.265} C_VEL
LIN {X 0,Y 438.768,Z 435.831,A -85,B 0,C 180,E1 -8949.843,E2 -8949.843} C_VEL
LIN {X 0,Y 439.111,Z 429.671,A -85,B 0,C 180,E1 -8951.409,E2 -8951.409} C_VEL
LIN {X 0,Y 439.504,Z 423.499,A -85,B 0,C 180,E1 -8952.656,E2 -8952.656} C_VEL
LIN {X 0,Y 440.061,Z 415.844,A -85,B 0,C 180,E1 -8953.921,E2 -8953.921} C_VEL
LIN {X 0,Y 440.551,Z 407.426,A -85,B 0,C 180,E1 -8955.063,E2 -8955.063} C_VEL
LIN {X 0,Y 441.143,Z 397.819,A -85,B 0,C 180,E1 -8956.127,E2 -8956.127} C_VEL
LIN {X 0,Y 441.74,Z 387.674,A -85,B 0,C 180,E1 -8957.04,E2 -8957.04} C_VEL
LIN {X 0,Y 442.338,Z 375.934,A -85,B 0,C 180,E1 -8957.882,E2 -8957.882} C_VEL
LIN {X 0,Y 442.793,Z 364.729,A -85,B 0,C 180,E1 -8958.498,E2 -8958.498} C_VEL
LIN {X 0,Y 443.206,Z 351.476,A -85,B 0,C 180,E1 -8959.019,E2 -8959.019} C_VEL
LIN {X 0,Y 443.49,Z 338.18,A -85,B 0,C 180,E1 -8959.346,E2 -8959.346} C_VEL
LIN {X 0,Y 444.407,Z 253.337,A -85,B 0,C 180,E1 -8960.769,E2 -8960.769} C_VEL
LIN {X 0,Y 440.878,Z 236.121,A -85,B 0,C 180,E1 -8961.238,E2 -8961.238} C_VEL
LIN {X 0,Y 440.907,Z 227.569,A -85,B 0,C 180,E1 -8962.967,E2 -8962.967} C_VEL
LIN {X 0,Y 439.39,Z 219.756,A -85,B 0,C 180,E1 -8964.658,E2 -8964.658} C_VEL
LIN {X 0,Y 439.337,Z 219.76,A -85,B 0,C 180,E1 -8968.145,E2 -8968.145} C_VEL
LIN {X 0,Y 439.391,Z 219.755,A -85,B 0,C 180,E1 -8971.332,E2 -8971.332} C_VEL
LIN {X 0,Y 439.374,Z 219.752,A -85,B 0,C 180,E1 -8974.421,E2 -8974.421} C_VEL
LIN {X 0,Y 439.336,Z 219.758,A -85,B 0,C 180,E1 -8977.43,E2 -8977.43} C_VEL
LIN {X 0,Y 439.415,Z 219.75,A -85,B 0,C 180,E1 -8980.668,E2 -8980.668} C_VEL
LIN {X 0,Y 439.439,Z 219.746,A -85,B 0,C 180,E1 -8984.23,E2 -8984.23} C_VEL
LIN {X 0,Y 439.488,Z 219.737,A -85,B 0,C 180,E1 -8988.007,E2 -8988.007} C_VEL
LIN {X 0,Y 439.487,Z 219.735,A -85,B 0,C 180,E1 -8991.731,E2 -8991.731} C_VEL
LIN {X 0,Y 439.596,Z 219.727,A -85,B 0,C 180,E1 -8994.501,E2 -8994.501} C_VEL
LIN {X 0,Y 439.621,Z 219.72,A -85,B 0,C 180,E1 -8998.173,E2 -8998.173} C_VEL
LIN {X 0,Y 439.746,Z 219.705,A -85,B 0,C 180,E1 -9000.005,E2 -9000.005} C_VEL
LIN {X 0,Y 439.601,Z 219.725,A -85,B 0,C 180,E1 -9002.754,E2 -9002.754} C_VEL
LIN {X 0,Y 439.588,Z 219.723,A -85,B 0,C 180,E1 -9006.43,E2 -9006.43} C_VEL
LIN {X 0,Y 439.479,Z 219.736,A -85,B 0,C 180,E1 -9009.207,E2 -9009.207} C_VEL
LIN {X 0,Y 439.462,Z 219.742,A -85,B 0,C 180,E1 -9012.942,E2 -9012.942} C_VEL
LIN {X 0,Y 439.444,Z 219.746,A -85,B 0,C 180,E1 -9016.352,E2 -9016.352} C_VEL
LIN {X 0,Y 439.401,Z 219.746,A -85,B 0,C 180,E1 -9019.631,E2 -9019.631} C_VEL
LIN {X 0,Y 439.362,Z 219.753,A -85,B 0,C 180,E1 -9022.58,E2 -9022.58} C_VEL
LIN {X 0,Y 439.354,Z 219.752,A -85,B 0,C 180,E1 -9025.592,E2 -9025.592} C_VEL
LIN {X 0,Y 439.393,Z 219.752,A -85,B 0,C 180,E1 -9028.679,E2 -9028.679} C_VEL
LIN {X 0,Y 439.366,Z 219.755,A -85,B 0,C 180,E1 -9032.032,E2 -9032.032} C_VEL
LIN {X 0,Y 439.39,Z 219.75,A -85,B 0,C 180,E1 -9035.342,E2 -9035.342} C_VEL
LIN {X 0,Y 439.353,Z 219.758,A -85,B 0,C 180,E1 -9038.602,E2 -9038.602} C_VEL
LIN {X 0,Y 439.35,Z 219.76,A -85,B 0,C 180,E1 -9042.214,E2 -9042.214} C_VEL
LIN {X 0,Y 439.374,Z 219.754,A -85,B 0,C 180,E1 -9045.269,E2 -9045.269} C_VEL
LIN {X 0,Y 439.365,Z 219.756,A -85,B 0,C 180,E1 -9048.751,E2 -9048.751} C_VEL
LIN {X 0,Y 439.357,Z 219.755,A -85,B 0,C 180,E1 -9051.615,E2 -9051.615} C_VEL
LIN {X 0,Y 439.393,Z 219.752,A -85,B 0,C 180,E1 -9054.845,E2 -9054.845} C_VEL
LIN {X 0,Y 439.354,Z 219.765,A -85,B 0,C 180,E1 -9058.139,E2 -9058.139} C_VEL
LIN {X 0,Y 439.386,Z 219.756,A -85,B 0,C 180,E1 -9061.325,E2 -9061.325} C_VEL
LIN {X 0,Y 439.369,Z 219.893,A -85,B 0,C 180,E1 -9063.169,E2 -9063.169} C_VEL
LIN {X 0,Y 441.747,Z 231.8,A -85,B 0,C 180,E1 -9065.567,E2 -9065.567} C_VEL
LIN {X 0,Y 441.972,Z 235.807,A -85,B 0,C 180,E1 -9066.328,E2 -9066.328} C_VEL
LIN {X 0,Y 441.087,Z 251.754,A -85,B 0,C 180,E1 -9069.237,E2 -9069.237} C_VEL
LIN {X 0,Y 440.473,Z 266.141,A -85,B 0,C 180,E1 -9071.796,E2 -9071.796} C_VEL
LIN {X 0,Y 444.081,Z 289.746,A -85,B 0,C 180,E1 -9072.365,E2 -9072.365} C_VEL
LIN {X 0,Y 443.249,Z 374.573,A -85,B 0,C 180,E1 -9073.802,E2 -9073.802} C_VEL
LIN {X 0,Y 442.728,Z 387.756,A -85,B 0,C 180,E1 -9074.197,E2 -9074.197} C_VEL
LIN {X 0,Y 442.164,Z 401.03,A -85,B 0,C 180,E1 -9074.796,E2 -9074.796} C_VEL
LIN {X 0,Y 441.534,Z 412.204,A -85,B 0,C 180,E1 -9075.482,E2 -9075.482} C_VEL
LIN {X 0,Y 440.943,Z 423.352,A -85,B 0,C 180,E1 -9076.359,E2 -9076.359} C_VEL
LIN {X 0,Y 440.295,Z 434.325,A -85,B 0,C 180,E1 -9077.439,E2 -9077.439} C_VEL
LIN {X 0,Y 439.806,Z 442.909,A -85,B 0,C 180,E1 -9078.478,E2 -9078.478} C_VEL
LIN {X 0,Y 439.228,Z 450.829,A -85,B 0,C 180,E1 -9079.63,E2 -9079.63} C_VEL
LIN {X 0,Y 438.865,Z 458.574,A -85,B 0,C 180,E1 -9081.018,E2 -9081.018} C_VEL
LIN {X 0,Y 438.538,Z 465.721,A -85,B 0,C 180,E1 -9082.634,E2 -9082.634} C_VEL
LIN {X 0,Y 438.365,Z 470.472,A -85,B 0,C 180,E1 -9084.017,E2 -9084.017} C_VEL
LIN {X 0,Y 438.344,Z 474.117,A -85,B 0,C 180,E1 -9085.402,E2 -9085.402} C_VEL
LIN {X 0,Y 438.286,Z 475.991,A -85,B 0,C 180,E1 -9086.323,E2 -9086.323} C_VEL
LIN {X 0,Y 438.346,Z 477.4,A -85,B 0,C 180,E1 -9087.243,E2 -9087.243} C_VEL
LIN {X 0,Y 438.301,Z 478.405,A -85,B 0,C 180,E1 -9088.162,E2 -9088.162} C_VEL
LIN {X 0,Y 438.26,Z 479.018,A -85,B 0,C 180,E1 -9089.081,E2 -9089.081} C_VEL
LIN {X 0,Y 438.261,Z 479.229,A -85,B 0,C 180,E1 -9090,E2 -9090} C_VEL
LIN {X 0,Y 438.301,Z 478.39,A -85,B 0,C 180,E1 -9091.838,E2 -9091.838} C_VEL
LIN {X 0,Y 438.346,Z 477.383,A -85,B 0,C 180,E1 -9092.757,E2 -9092.757} C_VEL
LIN {X 0,Y 438.286,Z 475.954,A -85,B 0,C 180,E1 -9093.677,E2 -9093.677} C_VEL
LIN {X 0,Y 438.382,Z 472.979,A -85,B 0,C 180,E1 -9095.059,E2 -9095.059} C_VEL
LIN {X 0,Y 438.46,Z 468.943,A -85,B 0,C 180,E1 -9096.442,E2 -9096.442} C_VEL
LIN {X 0,Y 438.674,Z 462.725,A -85,B 0,C 180,E1 -9098.058,E2 -9098.058} C_VEL
LIN {X 0,Y 438.966,Z 455.944,A -85,B 0,C 180,E1 -9099.445,E2 -9099.445} C_VEL
LIN {X 0,Y 439.399,Z 447.522,A -85,B 0,C 180,E1 -9100.832,E2 -9100.832} C_VEL
LIN {X 0,Y 439.989,Z 438.846,A -85,B 0,C 180,E1 -9101.984,E2 -9101.984} C_VEL
LIN {X 0,Y 440.533,Z 429.097,A -85,B 0,C 180,E1 -9103.046,E2 -9103.046} C_VEL
LIN {X 0,Y 441.16,Z 417.536,A -85,B 0,C 180,E1 -9104.06,E2 -9104.06} C_VEL
LIN {X 0,Y 441.739,Z 405.726,A -85,B 0,C 180,E1 -9104.865,E2 -9104.865} C_VEL
LIN {X 0,Y 442.346,Z 393.466,A -85,B 0,C 180,E1 -9105.492,E2 -9105.492} C_VEL
LIN {X 0,Y 442.838,Z 380.052,A -85,B 0,C 180,E1 -9105.977,E2 -9105.977} C_VEL
LIN {X 0,Y 443.113,Z 366.649,A -85,B 0,C 180,E1 -9106.262,E2 -9106.262} C_VEL
LIN {X 0,Y 443.828,Z 288.896,A -85,B 0,C 180,E1 -9107.555,E2 -9107.555} C_VEL
LIN {X 0,Y 440.405,Z 266.584,A -85,B 0,C 180,E1 -9108.082,E2 -9108.082} C_VEL
LIN {X 0,Y 441.316,Z 249.395,A -85,B 0,C 180,E1 -9111.241,E2 -9111.241} C_VEL
LIN {X 0,Y 442.094,Z 235.044,A -85,B 0,C 180,E1 -9113.914,E2 -9113.914} C_VEL
LIN {X 0,Y 441.293,Z 229.078,A -85,B 0,C 180,E1 -9115.096,E2 -9115.096} C_VEL
LIN {X 0,Y 439.375,Z 219.756,A -85,B 0,C 180,E1 -9117.056,E2 -9117.056} C_VEL
LIN {X 0,Y 439.37,Z 219.756,A -85,B 0,C 180,E1 -9120.254,E2 -9120.254} C_VEL
LIN {X 0,Y 439.348,Z 219.76,A -85,B 0,C 180,E1 -9123.71,E2 -9123.71} C_VEL
LIN {X 0,Y 439.332,Z 219.755,A -85,B 0,C 180,E1 -9126.88,E2 -9126.88} C_VEL
LIN {X 0,Y 439.355,Z 219.76,A -85,B 0,C 180,E1 -9129.838,E2 -9129.838} C_VEL
LIN {X 0,Y 439.325,Z 219.756,A -85,B 0,C 180,E1 -9132.615,E2 -9132.615} C_VEL
LIN {X 0,Y 439.363,Z 219.754,A -85,B 0,C 180,E1 -9135.262,E2 -9135.262} C_VEL
LIN {X 0,Y 439.363,Z 219.751,A -85,B 0,C 180,E1 -9138.745,E2 -9138.745} C_VEL
LIN {X 0,Y 439.353,Z 219.759,A -85,B 0,C 180,E1 -9141.609,E2 -9141.609} C_VEL
LIN {X 0,Y 439.349,Z 219.753,A -85,B 0,C 180,E1 -9144.835,E2 -9144.835} C_VEL
LIN {X 0,Y 439.348,Z 219.756,A -85,B 0,C 180,E1 -9148.134,E2 -9148.134} C_VEL
LIN {X 0,Y 439.379,Z 219.753,A -85,B 0,C 180,E1 -9151.32,E2 -9151.32} C_VEL
LIN {X 0,Y 439.344,Z 219.754,A -85,B 0,C 180,E1 -9154.407,E2 -9154.407} C_VEL
LIN {X 0,Y 439.361,Z 219.757,A -85,B 0,C 180,E1 -9157.42,E2 -9157.42} C_VEL
LIN {X 0,Y 439.385,Z 219.749,A -85,B 0,C 180,E1 -9160.68,E2 -9160.68} C_VEL
LIN {X 0,Y 439.442,Z 219.743,A -85,B 0,C 180,E1 -9164.219,E2 -9164.219} C_VEL
LIN {X 0,Y 439.466,Z 219.741,A -85,B 0,C 180,E1 -9167.996,E2 -9167.996} C_VEL
LIN {X 0,Y 439.472,Z 219.744,A -85,B 0,C 180,E1 -9171.72,E2 -9171.72} C_VEL
LIN {X 0,Y 439.586,Z 219.724,A -85,B 0,C 180,E1 -9174.49,E2 -9174.49} C_VEL
LIN {X 0,Y 439.61,Z 219.722,A -85,B 0,C 180,E1 -9178.163,E2 -9178.163} C_VEL
LIN {X 0,Y 439.635,Z 219.72,A -85,B 0,C 180,E1 -9179.995,E2 -9179.995} C_VEL
LIN {X 0,Y 439.599,Z 219.723,A -85,B 0,C 180,E1 -9182.744,E2 -9182.744} C_VEL
LIN {X 0,Y 439.533,Z 219.73,A -85,B 0,C 180,E1 -9186.421,E2 -9186.421} C_VEL
LIN {X 0,Y 439.459,Z 219.744,A -85,B 0,C 180,E1 -9189.197,E2 -9189.197} C_VEL
LIN {X 0,Y 439.444,Z 219.743,A -85,B 0,C 180,E1 -9192.932,E2 -9192.932} C_VEL
LIN {X 0,Y 439.422,Z 219.744,A -85,B 0,C 180,E1 -9196.342,E2 -9196.342} C_VEL
LIN {X 0,Y 439.375,Z 219.755,A -85,B 0,C 180,E1 -9199.621,E2 -9199.621} C_VEL
LIN {X 0,Y 439.332,Z 219.756,A -85,B 0,C 180,E1 -9202.57,E2 -9202.57} C_VEL
LIN {X 0,Y 439.347,Z 219.759,A -85,B 0,C 180,E1 -9205.581,E2 -9205.581} C_VEL
LIN {X 0,Y 439.383,Z 219.75,A -85,B 0,C 180,E1 -9208.668,E2 -9208.668} C_VEL
LIN {X 0,Y 439.332,Z 219.756,A -85,B 0,C 180,E1 -9212.025,E2 -9212.025} C_VEL
LIN {X 0,Y 439.354,Z 219.761,A -85,B 0,C 180,E1 -9215.335,E2 -9215.335} C_VEL
LIN {X 0,Y 439.34,Z 219.755,A -85,B 0,C 180,E1 -9218.59,E2 -9218.59} C_VEL
LIN {X 0,Y 439.344,Z 219.761,A -85,B 0,C 180,E1 -9221.252,E2 -9221.252} C_VEL
LIN {X 0,Y 439.357,Z 219.754,A -85,B 0,C 180,E1 -9224.724,E2 -9224.724} C_VEL
LIN {X 0,Y 439.346,Z 219.755,A -85,B 0,C 180,E1 -9227.791,E2 -9227.791} C_VEL
LIN {X 0,Y 439.376,Z 219.75,A -85,B 0,C 180,E1 -9230.223,E2 -9230.223} C_VEL
LIN {X 0,Y 439.325,Z 219.758,A -85,B 0,C 180,E1 -9233.709,E2 -9233.709} C_VEL
LIN {X 0,Y 439.318,Z 219.763,A -85,B 0,C 180,E1 -9237.05,E2 -9237.05} C_VEL
LIN {X 0,Y 439.339,Z 219.755,A -85,B 0,C 180,E1 -9240.272,E2 -9240.272} C_VEL
LIN {X 0,Y 439.372,Z 219.755,A -85,B 0,C 180,E1 -9243.393,E2 -9243.393} C_VEL
LIN {X 0,Y 439.339,Z 219.755,A -85,B 0,C 180,E1 -9246.427,E2 -9246.427} C_VEL
LIN {X 0,Y 439.353,Z 219.757,A -85,B 0,C 180,E1 -9249.396,E2 -9249.396} C_VEL
LIN {X 0,Y 439.376,Z 219.75,A -85,B 0,C 180,E1 -9252.308,E2 -9252.308} C_VEL
LIN {X 0,Y 439.39,Z 219.755,A -85,B 0,C 180,E1 -9255.172,E2 -9255.172} C_VEL
LIN {X 0,Y 439.45,Z 219.741,A -85,B 0,C 180,E1 -9258.001,E2 -9258.001} C_VEL
LIN {X 0,Y 439.49,Z 219.737,A -85,B 0,C 180,E1 -9261.725,E2 -9261.725} C_VEL
LIN {X 0,Y 439.567,Z 219.727,A -85,B 0,C 180,E1 -9264.495,E2 -9264.495} C_VEL
LIN {X 0,Y 439.572,Z 219.725,A -85,B 0,C 180,E1 -9268.168,E2 -9268.168} C_VEL
LIN {X 0,Y 439.699,Z 219.71,A -85,B 0,C 180,E1 -9270,E2 -9270} C_VEL
LIN {X 0,Y 439.591,Z 219.729,A -85,B 0,C 180,E1 -9270.942,E2 -9270.942} C_VEL
LIN {X 0,Y 438.853,Z 219.817,A -85,B 0,C 180,E1 -9271.707,E2 -9271.707} C_VEL
LIN {X 0,Y 435.862,Z 220.195,A -85,B 0,C 180,E1 -9272.945,E2 -9272.945} C_VEL
LIN {X 0,Y 433.412,Z 220.498,A -85,B 0,C 180,E1 -9273.946,E2 -9273.946} C_VEL
LIN {X 0,Y 432.439,Z 220.618,A -85,B 0,C 180,E1 -9274.72,E2 -9274.72} C_VEL
LIN {X 0,Y 432.401,Z 220.621,A -85,B 0,C 180,E1 -9274.982,E2 -9274.982} C_VEL
LIN {X 0,Y 432.522,Z 220.607,A -85,B 0,C 180,E1 -9277.68,E2 -9277.68} C_VEL
LIN {X 0,Y 432.413,Z 220.803,A -85,B 0,C 180,E1 -9281.187,E2 -9281.187} C_VEL
LIN {X 0,Y 433.846,Z 229.039,A -85,B 0,C 180,E1 -9283.108,E2 -9283.108} C_VEL
LIN {X 0,Y 433.776,Z 236.567,A -85,B 0,C 180,E1 -9284.724,E2 -9284.724} C_VEL
LIN {X 0,Y 437.391,Z 254.759,A -85,B 0,C 180,E1 -9285.194,E2 -9285.194} C_VEL
LIN {X 0,Y 436.294,Z 343.35,A -85,B 0,C 180,E1 -9286.704,E2 -9286.704} C_VEL
LIN {X 0,Y 435.937,Z 356.539,A -85,B 0,C 180,E1 -9287.11,E2 -9287.11} C_VEL
LIN {X 0,Y 435.533,Z 369.167,A -85,B 0,C 180,E1 -9287.691,E2 -9287.691} C_VEL
LIN {X 0,Y 434.966,Z 381.801,A -85,B 0,C 180,E1 -9288.487,E2 -9288.487} C_VEL
LIN {X 0,Y 434.394,Z 392.645,A -85,B 0,C 180,E1 -9289.369,E2 -9289.369} C_VEL
LIN {X 0,Y 433.738,Z 403.121,A -85,B 0,C 180,E1 -9290.429,E2 -9290.429} C_VEL
LIN {X 0,Y 433.189,Z 411.051,A -85,B 0,C 180,E1 -9291.409,E2 -9291.409} C_VEL
LIN {X 0,Y 432.629,Z 420.012,A -85,B 0,C 180,E1 -9292.756,E2 -9292.756} C_VEL
LIN {X 0,Y 432.218,Z 426.673,A -85,B 0,C 180,E1 -9293.985,E2 -9293.985} C_VEL
LIN {X 0,Y 431.806,Z 433.476,A -85,B 0,C 180,E1 -9295.55,E2 -9295.55} C_VEL
LIN {X 0,Y 431.534,Z 438.788,A -85,B 0,C 180,E1 -9297.129,E2 -9297.129} C_VEL
LIN {X 0,Y 431.414,Z 442.041,A -85,B 0,C 180,E1 -9298.412,E2 -9298.412} C_VEL
LIN {X 0,Y 431.266,Z 443.766,A -85,B 0,C 180,E1 -9299.266,E2 -9299.266} C_VEL
LIN {X 0,Y 431.163,Z 445.407,A -85,B 0,C 180,E1 -9300.351,E2 -9300.351} C_VEL
LIN {X 0,Y 431.061,Z 446.89,A -85,B 0,C 180,E1 -9302.042,E2 -9302.042} C_VEL
LIN {X 0,Y 431.063,Z 447.079,A -85,B 0,C 180,E1 -9303.762,E2 -9303.762} C_VEL
LIN {X 0,Y 431.122,Z 445.968,A -85,B 0,C 180,E1 -9305.418,E2 -9305.418} C_VEL
LIN {X 0,Y 431.309,Z 443.561,A -85,B 0,C 180,E1 -9307.077,E2 -9307.077} C_VEL
LIN {X 0,Y 431.525,Z 440.195,A -85,B 0,C 180,E1 -9308.592,E2 -9308.592} C_VEL
LIN {X 0,Y 431.747,Z 435.634,A -85,B 0,C 180,E1 -9310.099,E2 -9310.099} C_VEL
LIN {X 0,Y 432.122,Z 429.817,A -85,B 0,C 180,E1 -9311.582,E2 -9311.582} C_VEL
LIN {X 0,Y 432.559,Z 422.639,A -85,B 0,C 180,E1 -9313.03,E2 -9313.03} C_VEL
LIN {X 0,Y 433.205,Z 413.667,A -85,B 0,C 180,E1 -9314.464,E2 -9314.464} C_VEL
LIN {X 0,Y 433.853,Z 404.312,A -85,B 0,C 180,E1 -9315.673,E2 -9315.673} C_VEL
LIN {X 0,Y 434.498,Z 394.42,A -85,B 0,C 180,E1 -9316.707,E2 -9316.707} C_VEL
LIN {X 0,Y 435.171,Z 383.083,A -85,B 0,C 180,E1 -9317.653,E2 -9317.653} C_VEL
LIN {X 0,Y 435.718,Z 371.483,A -85,B 0,C 180,E1 -9318.414,E2 -9318.414} C_VEL
LIN {X 0,Y 436.194,Z 359.169,A -85,B 0,C 180,E1 -9319.017,E2 -9319.017} C_VEL
LIN {X 0,Y 436.599,Z 346.378,A -85,B 0,C 180,E1 -9319.441,E2 -9319.441} C_VEL
LIN {X 0,Y 436.856,Z 327.989,A -85,B 0,C 180,E1 -9319.796,E2 -9319.796} C_VEL
LIN {X 0,Y 437.606,Z 253.843,A -85,B 0,C 180,E1 -9321.066,E2 -9321.066} C_VEL
LIN {X 0,Y 433.961,Z 236.417,A -85,B 0,C 180,E1 -9321.548,E2 -9321.548} C_VEL
LIN {X 0,Y 433.914,Z 228.423,A -85,B 0,C 180,E1 -9323.191,E2 -9323.191} C_VEL
LIN {X 0,Y 432.341,Z 220.633,A -85,B 0,C 180,E1 -9324.906,E2 -9324.906} C_VEL
LIN {X 0,Y 432.288,Z 220.64,A -85,B 0,C 180,E1 -9327.712,E2 -9327.712} C_VEL
LIN {X 0,Y 432.318,Z 220.636,A -85,B 0,C 180,E1 -9330.819,E2 -9330.819} C_VEL
LIN {X 0,Y 432.333,Z 220.628,A -85,B 0,C 180,E1 -9333.973,E2 -9333.973} C_VEL
LIN {X 0,Y 432.29,Z 220.641,A -85,B 0,C 180,E1 -9337.041,E2 -9337.041} C_VEL
LIN {X 0,Y 432.36,Z 220.628,A -85,B 0,C 180,E1 -9340.52,E2 -9340.52} C_VEL
LIN {X 0,Y 432.407,Z 220.621,A -85,B 0,C 180,E1 -9343.967,E2 -9343.967} C_VEL
LIN {X 0,Y 432.461,Z 220.612,A -85,B 0,C 180,E1 -9347.81,E2 -9347.81} C_VEL
LIN {X 0,Y 432.447,Z 220.613,A -85,B 0,C 180,E1 -9351.595,E2 -9351.595} C_VEL
LIN {X 0,Y 432.572,Z 220.601,A -85,B 0,C 180,E1 -9354.411,E2 -9354.411} C_VEL
LIN {X 0,Y 432.591,Z 220.595,A -85,B 0,C 180,E1 -9358.143,E2 -9358.143} C_VEL
LIN {X 0,Y 432.716,Z 220.581,A -85,B 0,C 180,E1 -9360.005,E2 -9360.005} C_VEL
LIN {X 0,Y 432.555,Z 220.603,A -85,B 0,C 180,E1 -9362.799,E2 -9362.799} C_VEL
LIN {X 0,Y 432.576,Z 220.594,A -85,B 0,C 180,E1 -9365.599,E2 -9365.599} C_VEL
LIN {X 0,Y 432.454,Z 220.617,A -85,B 0,C 180,E1 -9368.415,E2 -9368.415} C_VEL
LIN {X 0,Y 432.454,Z 220.615,A -85,B 0,C 180,E1 -9372.201,E2 -9372.201} C_VEL
LIN {X 0,Y 432.427,Z 220.617,A -85,B 0,C 180,E1 -9376.043,E2 -9376.043} C_VEL
LIN {X 0,Y 432.386,Z 220.62,A -85,B 0,C 180,E1 -9379.489,E2 -9379.489} C_VEL
LIN {X 0,Y 432.309,Z 220.632,A -85,B 0,C 180,E1 -9382.969,E2 -9382.969} C_VEL
LIN {X 0,Y 432.307,Z 220.632,A -85,B 0,C 180,E1 -9386.04,E2 -9386.04} C_VEL
LIN {X 0,Y 432.329,Z 220.627,A -85,B 0,C 180,E1 -9389.193,E2 -9389.193} C_VEL
LIN {X 0,Y 432.321,Z 220.635,A -85,B 0,C 180,E1 -9392.447,E2 -9392.447} C_VEL
LIN {X 0,Y 432.337,Z 220.63,A -85,B 0,C 180,E1 -9395.822,E2 -9395.822} C_VEL
LIN {X 0,Y 432.317,Z 220.633,A -85,B 0,C 180,E1 -9398.713,E2 -9398.713} C_VEL
LIN {X 0,Y 432.306,Z 220.635,A -85,B 0,C 180,E1 -9401.804,E2 -9401.804} C_VEL
LIN {X 0,Y 432.339,Z 220.635,A -85,B 0,C 180,E1 -9404.351,E2 -9404.351} C_VEL
LIN {X 0,Y 432.288,Z 220.637,A -85,B 0,C 180,E1 -9407.024,E2 -9407.024} C_VEL
LIN {X 0,Y 432.296,Z 220.637,A -85,B 0,C 180,E1 -9409.831,E2 -9409.831} C_VEL
LIN {X 0,Y 432.3,Z 220.635,A -85,B 0,C 180,E1 -9413.023,E2 -9413.023} C_VEL
LIN {X 0,Y 432.338,Z 220.635,A -85,B 0,C 180,E1 -9416.005,E2 -9416.005} C_VEL
LIN {X 0,Y 432.34,Z 220.634,A -85,B 0,C 180,E1 -9419.496,E2 -9419.496} C_VEL
LIN {X 0,Y 432.314,Z 220.635,A -85,B 0,C 180,E1 -9422.858,E2 -9422.858} C_VEL
LIN {X 0,Y 434.765,Z 232.931,A -85,B 0,C 180,E1 -9425.403,E2 -9425.403} C_VEL
LIN {X 0,Y 435.074,Z 236.937,A -85,B 0,C 180,E1 -9426.182,E2 -9426.182} C_VEL
LIN {X 0,Y 434.055,Z 255.467,A -85,B 0,C 180,E1 -9429.617,E2 -9429.617} C_VEL
LIN {X 0,Y 433.556,Z 265.635,A -85,B 0,C 180,E1 -9431.474,E2 -9431.474} C_VEL
LIN {X 0,Y 437.329,Z 290.062,A -85,B 0,C 180,E1 -9432.077,E2 -9432.077} C_VEL
LIN {X 0,Y 436.449,Z 374.681,A -85,B 0,C 180,E1 -9433.543,E2 -9433.543} C_VEL
LIN {X 0,Y 435.878,Z 388.477,A -85,B 0,C 180,E1 -9433.972,E2 -9433.972} C_VEL
LIN {X 0,Y 435.313,Z 400.908,A -85,B 0,C 180,E1 -9434.551,E2 -9434.551} C_VEL
LIN {X 0,Y 434.668,Z 412.03,A -85,B 0,C 180,E1 -9435.247,E2 -9435.247} C_VEL
LIN {X 0,Y 434.047,Z 422.996,A -85,B 0,C 180,E1 -9436.123,E2 -9436.123} C_VEL
LIN {X 0,Y 433.313,Z 434.12,A -85,B 0,C 180,E1 -9437.233,E2 -9437.233} C_VEL
LIN {X 0,Y 432.821,Z 442.695,A -85,B 0,C 180,E1 -9438.29,E2 -9438.29} C_VEL
LIN {X 0,Y 432.214,Z 450.607,A -85,B 0,C 180,E1 -9439.46,E2 -9439.46} C_VEL
LIN {X 0,Y 431.805,Z 458.342,A -85,B 0,C 180,E1 -9440.869,E2 -9440.869} C_VEL
LIN {X 0,Y 431.469,Z 465.486,A -85,B 0,C 180,E1 -9442.513,E2 -9442.513} C_VEL
LIN {X 0,Y 431.265,Z 470.663,A -85,B 0,C 180,E1 -9444.06,E2 -9444.06} C_VEL
LIN {X 0,Y 431.273,Z 473.874,A -85,B 0,C 180,E1 -9445.327,E2 -9445.327} C_VEL
LIN {X 0,Y 431.193,Z 475.742,A -85,B 0,C 180,E1 -9446.262,E2 -9446.262} C_VEL
LIN {X 0,Y 431.242,Z 477.147,A -85,B 0,C 180,E1 -9447.198,E2 -9447.198} C_VEL
LIN {X 0,Y 431.224,Z 478.15,A -85,B 0,C 180,E1 -9448.132,E2 -9448.132} C_VEL
LIN {X 0,Y 431.177,Z 478.761,A -85,B 0,C 180,E1 -9449.066,E2 -9449.066} C_VEL
LIN {X 0,Y 431.175,Z 478.966,A -85,B 0,C 180,E1 -9450,E2 -9450} C_VEL
LIN {X 0,Y 431.224,Z 478.119,A -85,B 0,C 180,E1 -9451.868,E2 -9451.868} C_VEL
LIN {X 0,Y 431.242,Z 477.107,A -85,B 0,C 180,E1 -9452.802,E2 -9452.802} C_VEL
LIN {X 0,Y 431.193,Z 475.67,A -85,B 0,C 180,E1 -9453.738,E2 -9453.738} C_VEL
LIN {X 0,Y 431.292,Z 472.686,A -85,B 0,C 180,E1 -9455.142,E2 -9455.142} C_VEL
LIN {X 0,Y 431.388,Z 468.64,A -85,B 0,C 180,E1 -9456.548,E2 -9456.548} C_VEL
LIN {X 0,Y 431.607,Z 462.405,A -85,B 0,C 180,E1 -9458.191,E2 -9458.191} C_VEL
LIN {X 0,Y 431.915,Z 455.609,A -85,B 0,C 180,E1 -9459.601,E2 -9459.601} C_VEL
LIN {X 0,Y 432.4,Z 447.165,A -85,B 0,C 180,E1 -9461.01,E2 -9461.01} C_VEL
LIN {X 0,Y 432.997,Z 438.463,A -85,B 0,C 180,E1 -9462.181,E2 -9462.181} C_VEL
LIN {X 0,Y 433.624,Z 428.185,A -85,B 0,C 180,E1 -9463.309,E2 -9463.309} C_VEL
LIN {X 0,Y 434.232,Z 417.093,A -85,B 0,C 180,E1 -9464.289,E2 -9464.289} C_VEL
LIN {X 0,Y 434.869,Z 405.212,A -85,B 0,C 180,E1 -9465.105,E2 -9465.105} C_VEL
LIN {X 0,Y 435.515,Z 392.878,A -85,B 0,C 180,E1 -9465.742,E2 -9465.742} C_VEL
LIN {X 0,Y 435.977,Z 380.264,A -85,B 0,C 180,E1 -9466.205,E2 -9466.205} C_VEL
LIN {X 0,Y 436.265,Z 367.261,A -85,B 0,C 180,E1 -9466.494,E2 -9466.494} C_VEL
LIN {X 0,Y 436.973,Z 289.408,A -85,B 0,C 180,E1 -9467.813,E2 -9467.813} C_VEL
LIN {X 0,Y 433.462,Z 266.259,A -85,B 0,C 180,E1 -9468.382,E2 -9468.382} C_VEL
LIN {X 0,Y 434.421,Z 249.078,A -85,B 0,C 180,E1 -9471.595,E2 -9471.595} C_VEL
LIN {X 0,Y 435.157,Z 236.038,A -85,B 0,C 180,E1 -9474.066,E2 -9474.066} C_VEL
LIN {X 0,Y 434.096,Z 229.321,A -85,B 0,C 180,E1 -9475.427,E2 -9475.427} C_VEL
LIN {X 0,Y 432.326,Z 220.634,A -85,B 0,C 180,E1 -9477.272,E2 -9477.272} C_VEL
LIN {X 0,Y 432.315,Z 220.633,A -85,B 0,C 180,E1 -9480.498,E2 -9480.498} C_VEL
LIN {X 0,Y 432.315,Z 220.635,A -85,B 0,C 180,E1 -9483.99,E2 -9483.99} C_VEL
LIN {X 0,Y 432.309,Z 220.632,A -85,B 0,C 180,E1 -9487.19,E2 -9487.19} C_VEL
LIN {X 0,Y 432.296,Z 220.635,A -85,B 0,C 180,E1 -9490.169,E2 -9490.169} C_VEL
LIN {X 0,Y 432.262,Z 220.637,A -85,B 0,C 180,E1 -9493.067,E2 -9493.067} C_VEL
LIN {X 0,Y 432.317,Z 220.636,A -85,B 0,C 180,E1 -9495.666,E2 -9495.666} C_VEL
LIN {X 0,Y 432.31,Z 220.631,A -85,B 0,C 180,E1 -9498.4,E2 -9498.4} C_VEL
LIN {X 0,Y 432.319,Z 220.635,A -85,B 0,C 180,E1 -9501.844,E2 -9501.844} C_VEL
LIN {X 0,Y 432.298,Z 220.635,A -85,B 0,C 180,E1 -9505.315,E2 -9505.315} C_VEL
LIN {X 0,Y 432.303,Z 220.631,A -85,B 0,C 180,E1 -9508.648,E2 -9508.648} C_VEL
LIN {X 0,Y 432.313,Z 220.635,A -85,B 0,C 180,E1 -9511.868,E2 -9511.868} C_VEL
LIN {X 0,Y 432.348,Z 220.632,A -85,B 0,C 180,E1 -9515.544,E2 -9515.544} C_VEL
LIN {X 0,Y 432.336,Z 220.628,A -85,B 0,C 180,E1 -9519.041,E2 -9519.041} C_VEL
LIN {X 0,Y 432.335,Z 220.63,A -85,B 0,C 180,E1 -9522.005,E2 -9522.005} C_VEL
LIN {X 0,Y 432.357,Z 220.625,A -85,B 0,C 180,E1 -9524.921,E2 -9524.921} C_VEL
LIN {X 0,Y 432.446,Z 220.618,A -85,B 0,C 180,E1 -9527.798,E2 -9527.798} C_VEL
LIN {X 0,Y 432.439,Z 220.622,A -85,B 0,C 180,E1 -9531.584,E2 -9531.584} C_VEL
LIN {X 0,Y 432.541,Z 220.601,A -85,B 0,C 180,E1 -9534.4,E2 -9534.4} C_VEL
LIN {X 0,Y 432.579,Z 220.598,A -85,B 0,C 180,E1 -9538.133,E2 -9538.133} C_VEL
LIN {X 0,Y 432.587,Z 220.598,A -85,B 0,C 180,E1 -9539.995,E2 -9539.995} C_VEL
LIN {X 0,Y 432.553,Z 220.601,A -85,B 0,C 180,E1 -9542.788,E2 -9542.788} C_VEL
LIN {X 0,Y 432.49,Z 220.608,A -85,B 0,C 180,E1 -9546.526,E2 -9546.526} C_VEL
LIN {X 0,Y 432.405,Z 220.625,A -85,B 0,C 180,E1 -9549.348,E2 -9549.348} C_VEL
LIN {X 0,Y 432.41,Z 220.619,A -85,B 0,C 180,E1 -9552.797,E2 -9552.797} C_VEL
LIN {X 0,Y 432.388,Z 220.62,A -85,B 0,C 180,E1 -9556.472,E2 -9556.472} C_VEL
LIN {X 0,Y 432.311,Z 220.632,A -85,B 0,C 180,E1 -9559.955,E2 -9559.955} C_VEL
LIN {X 0,Y 432.286,Z 220.636,A -85,B 0,C 180,E1 -9562.959,E2 -9562.959} C_VEL
LIN {X 0,Y 432.306,Z 220.634,A -85,B 0,C 180,E1 -9564.997,E2 -9564.997} C_VEL
LIN {X 0,Y 432.347,Z 220.626,A -85,B 0,C 180,E1 -9568.118,E2 -9568.118} C_VEL
LIN {X 0,Y 432.284,Z 220.641,A -85,B 0,C 180,E1 -9571.341,E2 -9571.341} C_VEL
LIN {X 0,Y 432.3,Z 220.632,A -85,B 0,C 180,E1 -9574.672,E2 -9574.672} C_VEL
LIN {X 0,Y 432.296,Z 220.632,A -85,B 0,C 180,E1 -9578.145,E2 -9578.145} C_VEL
LIN {X 0,Y 432.288,Z 220.637,A -85,B 0,C 180,E1 -9581.597,E2 -9581.597} C_VEL
LIN {X 0,Y 432.293,Z 220.632,A -85,B 0,C 180,E1 -9584.342,E2 -9584.342} C_VEL
LIN {X 0,Y 432.272,Z 220.639,A -85,B 0,C 180,E1 -9587.011,E2 -9587.011} C_VEL
LIN {X 0,Y 432.283,Z 220.635,A -85,B 0,C 180,E1 -9589.817,E2 -9589.817} C_VEL
LIN {X 0,Y 432.263,Z 220.641,A -85,B 0,C 180,E1 -9593.019,E2 -9593.019} C_VEL
LIN {X 0,Y 432.305,Z 220.631,A -85,B 0,C 180,E1 -9595.993,E2 -9595.993} C_VEL
LIN {X 0,Y 432.338,Z 220.628,A -85,B 0,C 180,E1 -9599.74,E2 -9599.74} C_VEL
LIN {X 0,Y 432.342,Z 220.631,A -85,B 0,C 180,E1 -9603.369,E2 -9603.369} C_VEL
LIN {X 0,Y 432.32,Z 220.629,A -85,B 0,C 180,E1 -9606.021,E2 -9606.021} C_VEL
LIN {X 0,Y 432.317,Z 220.636,A -85,B 0,C 180,E1 -9609.045,E2 -9609.045} C_VEL
LIN {X 0,Y 432.321,Z 220.629,A -85,B 0,C 180,E1 -9612.009,E2 -9612.009} C_VEL
LIN {X 0,Y 432.34,Z 220.632,A -85,B 0,C 180,E1 -9614.925,E2 -9614.925} C_VEL
LIN {X 0,Y 432.421,Z 220.617,A -85,B 0,C 180,E1 -9617.803,E2 -9617.803} C_VEL
LIN {X 0,Y 432.434,Z 220.617,A -85,B 0,C 180,E1 -9621.589,E2 -9621.589} C_VEL
LIN {X 0,Y 432.544,Z 220.602,A -85,B 0,C 180,E1 -9624.406,E2 -9624.406} C_VEL
LIN {X 0,Y 432.543,Z 220.601,A -85,B 0,C 180,E1 -9628.138,E2 -9628.138} C_VEL
LIN {X 0,Y 432.67,Z 220.585,A -85,B 0,C 180,E1 -9630,E2 -9630} C_VEL
LIN {X 0,Y 432.55,Z 220.605,A -85,B 0,C 180,E1 -9632.794,E2 -9632.794} C_VEL
LIN {X 0,Y 432.401,Z 220.621,A -85,B 0,C 180,E1 -9634.982,E2 -9634.982} C_VEL
LIN {X 0,Y 431.843,Z 220.693,A -85,B 0,C 180,E1 -9635.761,E2 -9635.761} C_VEL
LIN {X 0,Y 429.012,Z 221.049,A -85,B 0,C 180,E1 -9637.026,E2 -9637.026} C_VEL
LIN {X 0,Y 426.537,Z 221.354,A -85,B 0,C 180,E1 -9638.047,E2 -9638.047} C_VEL
LIN {X 0,Y 425.454,Z 221.492,A -85,B 0,C 180,E1 -9638.837,E2 -9638.837} C_VEL
LIN {X 0,Y 425.359,Z 221.5,A -85,B 0,C 180,E1 -9639.105,E2 -9639.105} C_VEL
LIN {X 0,Y 425.347,Z 221.569,A -85,B 0,C 180,E1 -9640.953,E2 -9640.953} C_VEL
LIN {X 0,Y 426.8,Z 229.53,A -85,B 0,C 180,E1 -9642.844,E2 -9642.844} C_VEL
LIN {X 0,Y 426.906,Z 234.489,A -85,B 0,C 180,E1 -9643.962,E2 -9643.962} C_VEL
LIN {X 0,Y 426.82,Z 236.564,A -85,B 0,C 180,E1 -9644.421,E2 -9644.421} C_VEL
LIN {X 0,Y 430.599,Z 255.515,A -85,B 0,C 180,E1 -9644.925,E2 -9644.925} C_VEL
LIN {X 0,Y 429.461,Z 343.786,A -85,B 0,C 180,E1 -9646.458,E2 -9646.458} C_VEL
LIN {X 0,Y 429.084,Z 357.688,A -85,B 0,C 180,E1 -9646.901,E2 -9646.901} C_VEL
LIN {X 0,Y 428.658,Z 369.733,A -85,B 0,C 180,E1 -9647.471,E2 -9647.471} C_VEL
LIN {X 0,Y 428.157,Z 380.831,A -85,B 0,C 180,E1 -9648.172,E2 -9648.172} C_VEL
LIN {X 0,Y 427.512,Z 391.935,A -85,B 0,C 180,E1 -9649.07,E2 -9649.07} C_VEL
LIN {X 0,Y 426.823,Z 403.179,A -85,B 0,C 180,E1 -9650.215,E2 -9650.215} C_VEL
LIN {X 0,Y 426.187,Z 411.605,A -85,B 0,C 180,E1 -9651.271,E2 -9651.271} C_VEL
LIN {X 0,Y 425.646,Z 420.205,A -85,B 0,C 180,E1 -9652.589,E2 -9652.589} C_VEL
LIN {X 0,Y 425.085,Z 428.364,A -85,B 0,C 180,E1 -9654.154,E2 -9654.154} C_VEL
LIN {X 0,Y 424.739,Z 433.893,A -85,B 0,C 180,E1 -9655.48,E2 -9655.48} C_VEL
LIN {X 0,Y 424.462,Z 439.189,A -85,B 0,C 180,E1 -9657.092,E2 -9657.092} C_VEL
LIN {X 0,Y 424.28,Z 443.065,A -85,B 0,C 180,E1 -9658.709,E2 -9658.709} C_VEL
LIN {X 0,Y 424.061,Z 445.882,A -85,B 0,C 180,E1 -9660.497,E2 -9660.497} C_VEL
LIN {X 0,Y 423.984,Z 447.287,A -85,B 0,C 180,E1 -9662.303,E2 -9662.303} C_VEL
LIN {X 0,Y 423.982,Z 447.244,A -85,B 0,C 180,E1 -9664.038,E2 -9664.038} C_VEL
LIN {X 0,Y 424.046,Z 445.95,A -85,B 0,C 180,E1 -9665.711,E2 -9665.711} C_VEL
LIN {X 0,Y 424.253,Z 443.473,A -85,B 0,C 180,E1 -9667.344,E2 -9667.344} C_VEL
LIN {X 0,Y 424.481,Z 439.707,A -85,B 0,C 180,E1 -9668.986,E2 -9668.986} C_VEL
LIN {X 0,Y 424.75,Z 435.153,A -85,B 0,C 180,E1 -9670.449,E2 -9670.449} C_VEL
LIN {X 0,Y 425.177,Z 429.118,A -85,B 0,C 180,E1 -9671.953,E2 -9671.953} C_VEL
LIN {X 0,Y 425.687,Z 421.676,A -85,B 0,C 180,E1 -9673.424,E2 -9673.424} C_VEL
LIN {X 0,Y 426.37,Z 412.502,A -85,B 0,C 180,E1 -9674.875,E2 -9674.875} C_VEL
LIN {X 0,Y 427.036,Z 403.5,A -85,B 0,C 180,E1 -9676.018,E2 -9676.018} C_VEL
LIN {X 0,Y 427.756,Z 392.438,A -85,B 0,C 180,E1 -9677.152,E2 -9677.152} C_VEL
LIN {X 0,Y 428.399,Z 381.628,A -85,B 0,C 180,E1 -9678.036,E2 -9678.036} C_VEL
LIN {X 0,Y 429.017,Z 369.566,A -85,B 0,C 180,E1 -9678.799,E2 -9678.799} C_VEL
LIN {X 0,Y 429.563,Z 356.205,A -85,B 0,C 180,E1 -9679.414,E2 -9679.414} C_VEL
LIN {X 0,Y 429.849,Z 343.699,A -85,B 0,C 180,E1 -9679.799,E2 -9679.799} C_VEL
LIN {X 0,Y 430.909,Z 254.851,A -85,B 0,C 180,E1 -9681.358,E2 -9681.358} C_VEL
LIN {X 0,Y 427.067,Z 236.609,A -85,B 0,C 180,E1 -9681.892,E2 -9681.892} C_VEL
LIN {X 0,Y 427.113,Z 230.828,A -85,B 0,C 180,E1 -9683.097,E2 -9683.097} C_VEL
LIN {X 0,Y 425.31,Z 221.51,A -85,B 0,C 180,E1 -9685.17,E2 -9685.17} C_VEL
LIN {X 0,Y 425.229,Z 221.518,A -85,B 0,C 180,E1 -9688.079,E2 -9688.079} C_VEL
LIN {X 0,Y 425.304,Z 221.509,A -85,B 0,C 180,E1 -9691.374,E2 -9691.374} C_VEL
LIN {X 0,Y 425.264,Z 221.511,A -85,B 0,C 180,E1 -9694.56,E2 -9694.56} C_VEL
LIN {X 0,Y 425.259,Z 221.51,A -85,B 0,C 180,E1 -9697.667,E2 -9697.667} C_VEL
LIN {X 0,Y 425.336,Z 221.505,A -85,B 0,C 180,E1 -9700.71,E2 -9700.71} C_VEL
LIN {X 0,Y 425.365,Z 221.499,A -85,B 0,C 180,E1 -9703.694,E2 -9703.694} C_VEL
LIN {X 0,Y 425.41,Z 221.491,A -85,B 0,C 180,E1 -9707.604,E2 -9707.604} C_VEL
LIN {X 0,Y 425.391,Z 221.492,A -85,B 0,C 180,E1 -9711.455,E2 -9711.455} C_VEL
LIN {X 0,Y 425.528,Z 221.478,A -85,B 0,C 180,E1 -9714.319,E2 -9714.319} C_VEL
LIN {X 0,Y 425.56,Z 221.471,A -85,B 0,C 180,E1 -9718.113,E2 -9718.113} C_VEL
LIN {X 0,Y 425.685,Z 221.457,A -85,B 0,C 180,E1 -9720.005,E2 -9720.005} C_VEL
LIN {X 0,Y 425.51,Z 221.48,A -85,B 0,C 180,E1 -9722.845,E2 -9722.845} C_VEL
LIN {X 0,Y 425.532,Z 221.471,A -85,B 0,C 180,E1 -9725.692,E2 -9725.692} C_VEL
LIN {X 0,Y 425.399,Z 221.498,A -85,B 0,C 180,E1 -9728.556,E2 -9728.556} C_VEL
LIN {X 0,Y 425.407,Z 221.495,A -85,B 0,C 180,E1 -9732.407,E2 -9732.407} C_VEL
LIN {X 0,Y 425.386,Z 221.497,A -85,B 0,C 180,E1 -9736.316,E2 -9736.316} C_VEL
LIN {X 0,Y 425.328,Z 221.499,A -85,B 0,C 180,E1 -9739.64,E2 -9739.64} C_VEL
LIN {X 0,Y 425.288,Z 221.506,A -85,B 0,C 180,E1 -9742.343,E2 -9742.343} C_VEL
LIN {X 0,Y 425.252,Z 221.509,A -85,B 0,C 180,E1 -9745.452,E2 -9745.452} C_VEL
LIN {X 0,Y 425.31,Z 221.504,A -85,B 0,C 180,E1 -9748.864,E2 -9748.864} C_VEL
LIN {X 0,Y 425.263,Z 221.511,A -85,B 0,C 180,E1 -9751.931,E2 -9751.931} C_VEL
LIN {X 0,Y 425.296,Z 221.506,A -85,B 0,C 180,E1 -9755.34,E2 -9755.34} C_VEL
LIN {X 0,Y 425.27,Z 221.509,A -85,B 0,C 180,E1 -9758.906,E2 -9758.906} C_VEL
LIN {X 0,Y 425.249,Z 221.516,A -85,B 0,C 180,E1 -9761.954,E2 -9761.954} C_VEL
LIN {X 0,Y 425.278,Z 221.51,A -85,B 0,C 180,E1 -9765.288,E2 -9765.288} C_VEL
LIN {X 0,Y 425.252,Z 221.516,A -85,B 0,C 180,E1 -9768.62,E2 -9768.62} C_VEL
LIN {X 0,Y 425.275,Z 221.513,A -85,B 0,C 180,E1 -9772.307,E2 -9772.307} C_VEL
LIN {X 0,Y 425.291,Z 221.511,A -85,B 0,C 180,E1 -9775.817,E2 -9775.817} C_VEL
LIN {X 0,Y 425.295,Z 221.512,A -85,B 0,C 180,E1 -9779.243,E2 -9779.243} C_VEL
LIN {X 0,Y 425.265,Z 221.515,A -85,B 0,C 180,E1 -9782.437,E2 -9782.437} C_VEL
LIN {X 0,Y 425.27,Z 221.621,A -85,B 0,C 180,E1 -9782.629,E2 -9782.629} C_VEL
LIN {X 0,Y 427.823,Z 234.076,A -85,B 0,C 180,E1 -9785.236,E2 -9785.236} C_VEL
LIN {X 0,Y 428.169,Z 238.084,A -85,B 0,C 180,E1 -9786.031,E2 -9786.031} C_VEL
LIN {X 0,Y 427.078,Z 256.805,A -85,B 0,C 180,E1 -9789.558,E2 -9789.558} C_VEL
LIN {X 0,Y 426.599,Z 265.293,A -85,B 0,C 180,E1 -9791.14,E2 -9791.14} C_VEL
LIN {X 0,Y 430.618,Z 290.841,A -85,B 0,C 180,E1 -9791.791,E2 -9791.791} C_VEL
LIN {X 0,Y 429.675,Z 374.906,A -85,B 0,C 180,E1 -9793.276,E2 -9793.276} C_VEL
LIN {X 0,Y 429.067,Z 388.533,A -85,B 0,C 180,E1 -9793.71,E2 -9793.71} C_VEL
LIN {X 0,Y 428.49,Z 400.86,A -85,B 0,C 180,E1 -9794.299,E2 -9794.299} C_VEL
LIN {X 0,Y 427.696,Z 413.512,A -85,B 0,C 180,E1 -9795.123,E2 -9795.123} C_VEL
LIN {X 0,Y 427.023,Z 424.49,A -85,B 0,C 180,E1 -9796.044,E2 -9796.044} C_VEL
LIN {X 0,Y 426.304,Z 434.981,A -85,B 0,C 180,E1 -9797.141,E2 -9797.141} C_VEL
LIN {X 0,Y 425.729,Z 444.171,A -85,B 0,C 180,E1 -9798.333,E2 -9798.333} C_VEL
LIN {X 0,Y 425.036,Z 453.138,A -85,B 0,C 180,E1 -9799.761,E2 -9799.761} C_VEL
LIN {X 0,Y 424.682,Z 460.367,A -85,B 0,C 180,E1 -9801.195,E2 -9801.195} C_VEL
LIN {X 0,Y 424.348,Z 466.954,A -85,B 0,C 180,E1 -9802.865,E2 -9802.865} C_VEL
LIN {X 0,Y 424.179,Z 471.315,A -85,B 0,C 180,E1 -9804.295,E2 -9804.295} C_VEL
LIN {X 0,Y 424.202,Z 473.631,A -85,B 0,C 180,E1 -9805.248,E2 -9805.248} C_VEL
LIN {X 0,Y 424.104,Z 475.492,A -85,B 0,C 180,E1 -9806.199,E2 -9806.199} C_VEL
LIN {X 0,Y 424.139,Z 476.894,A -85,B 0,C 180,E1 -9807.151,E2 -9807.151} C_VEL
LIN {X 0,Y 424.149,Z 477.897,A -85,B 0,C 180,E1 -9808.101,E2 -9808.101} C_VEL
LIN {X 0,Y 424.097,Z 478.504,A -85,B 0,C 180,E1 -9809.051,E2 -9809.051} C_VEL
LIN {X 0,Y 424.093,Z 478.702,A -85,B 0,C 180,E1 -9810,E2 -9810} C_VEL
LIN {X 0,Y 424.149,Z 477.848,A -85,B 0,C 180,E1 -9811.899,E2 -9811.899} C_VEL
LIN {X 0,Y 424.139,Z 476.831,A -85,B 0,C 180,E1 -9812.849,E2 -9812.849} C_VEL
LIN {X 0,Y 424.105,Z 475.385,A -85,B 0,C 180,E1 -9813.801,E2 -9813.801} C_VEL
LIN {X 0,Y 424.204,Z 472.393,A -85,B 0,C 180,E1 -9815.228,E2 -9815.228} C_VEL
LIN {X 0,Y 424.311,Z 468.335,A -85,B 0,C 180,E1 -9816.658,E2 -9816.658} C_VEL
LIN {X 0,Y 424.54,Z 462.085,A -85,B 0,C 180,E1 -9818.328,E2 -9818.328} C_VEL
LIN {X 0,Y 424.888,Z 455.275,A -85,B 0,C 180,E1 -9819.761,E2 -9819.761} C_VEL
LIN {X 0,Y 425.405,Z 446.807,A -85,B 0,C 180,E1 -9821.193,E2 -9821.193} C_VEL
LIN {X 0,Y 426.015,Z 438.08,A -85,B 0,C 180,E1 -9822.384,E2 -9822.384} C_VEL
LIN {X 0,Y 426.684,Z 427.583,A -85,B 0,C 180,E1 -9823.549,E2 -9823.549} C_VEL
LIN {X 0,Y 427.318,Z 416.649,A -85,B 0,C 180,E1 -9824.525,E2 -9824.525} C_VEL
LIN {X 0,Y 427.992,Z 404.699,A -85,B 0,C 180,E1 -9825.354,E2 -9825.354} C_VEL
LIN {X 0,Y 428.667,Z 392.288,A -85,B 0,C 180,E1 -9826,E2 -9826} C_VEL
LIN {X 0,Y 429.174,Z 379.521,A -85,B 0,C 180,E1 -9826.469,E2 -9826.469} C_VEL
LIN {X 0,Y 429.431,Z 366.114,A -85,B 0,C 180,E1 -9826.765,E2 -9826.765} C_VEL
LIN {X 0,Y 430.211,Z 290.357,A -85,B 0,C 180,E1 -9828.068,E2 -9828.068} C_VEL
LIN {X 0,Y 426.495,Z 266.035,A -85,B 0,C 180,E1 -9828.673,E2 -9828.673} C_VEL
LIN {X 0,Y 427.514,Z 248.752,A -85,B 0,C 180,E1 -9831.961,E2 -9831.961} C_VEL
LIN {X 0,Y 428.21,Z 237.009,A -85,B 0,C 180,E1 -9834.224,E2 -9834.224} C_VEL
LIN {X 0,Y 426.557,Z 227.758,A -85,B 0,C 180,E1 -9836.15,E2 -9836.15} C_VEL
LIN {X 0,Y 425.293,Z 221.511,A -85,B 0,C 180,E1 -9837.516,E2 -9837.516} C_VEL
LIN {X 0,Y 425.256,Z 221.512,A -85,B 0,C 180,E1 -9840.818,E2 -9840.818} C_VEL
LIN {X 0,Y 425.272,Z 221.509,A -85,B 0,C 180,E1 -9844.276,E2 -9844.276} C_VEL
LIN {X 0,Y 425.273,Z 221.513,A -85,B 0,C 180,E1 -9847.694,E2 -9847.694} C_VEL
LIN {X 0,Y 425.252,Z 221.512,A -85,B 0,C 180,E1 -9851.38,E2 -9851.38} C_VEL
LIN {X 0,Y 425.267,Z 221.51,A -85,B 0,C 180,E1 -9855.284,E2 -9855.284} C_VEL
LIN {X 0,Y 425.251,Z 221.51,A -85,B 0,C 180,E1 -9858.614,E2 -9858.614} C_VEL
LIN {X 0,Y 425.269,Z 221.508,A -85,B 0,C 180,E1 -9862.301,E2 -9862.301} C_VEL
LIN {X 0,Y 425.272,Z 221.513,A -85,B 0,C 180,E1 -9865.81,E2 -9865.81} C_VEL
LIN {X 0,Y 425.289,Z 221.507,A -85,B 0,C 180,E1 -9869.237,E2 -9869.237} C_VEL
LIN {X 0,Y 425.294,Z 221.508,A -85,B 0,C 180,E1 -9871.361,E2 -9871.361} C_VEL
LIN {X 0,Y 425.246,Z 221.51,A -85,B 0,C 180,E1 -9874.547,E2 -9874.547} C_VEL
LIN {X 0,Y 425.288,Z 221.512,A -85,B 0,C 180,E1 -9877.657,E2 -9877.657} C_VEL
LIN {X 0,Y 425.323,Z 221.5,A -85,B 0,C 180,E1 -9880.698,E2 -9880.698} C_VEL
LIN {X 0,Y 425.371,Z 221.501,A -85,B 0,C 180,E1 -9883.683,E2 -9883.683} C_VEL
LIN {X 0,Y 425.402,Z 221.498,A -85,B 0,C 180,E1 -9887.593,E2 -9887.593} C_VEL
LIN {X 0,Y 425.387,Z 221.499,A -85,B 0,C 180,E1 -9891.444,E2 -9891.444} C_VEL
LIN {X 0,Y 425.5,Z 221.479,A -85,B 0,C 180,E1 -9894.307,E2 -9894.307} C_VEL
LIN {X 0,Y 425.549,Z 221.474,A -85,B 0,C 180,E1 -9898.102,E2 -9898.102} C_VEL
LIN {X 0,Y 425.423,Z 221.49,A -85,B 0,C 180,E1 -9900.941,E2 -9900.941} C_VEL
LIN {X 0,Y 425.508,Z 221.478,A -85,B 0,C 180,E1 -9902.835,E2 -9902.835} C_VEL
LIN {X 0,Y 425.452,Z 221.485,A -85,B 0,C 180,E1 -9906.634,E2 -9906.634} C_VEL
LIN {X 0,Y 425.366,Z 221.502,A -85,B 0,C 180,E1 -9909.504,E2 -9909.504} C_VEL
LIN {X 0,Y 425.373,Z 221.496,A -85,B 0,C 180,E1 -9912.897,E2 -9912.897} C_VEL
LIN {X 0,Y 425.337,Z 221.499,A -85,B 0,C 180,E1 -9916.598,E2 -9916.598} C_VEL
LIN {X 0,Y 425.302,Z 221.508,A -85,B 0,C 180,E1 -9919.629,E2 -9919.629} C_VEL
LIN {X 0,Y 425.273,Z 221.514,A -85,B 0,C 180,E1 -9923.36,E2 -9923.36} C_VEL
LIN {X 0,Y 425.275,Z 221.507,A -85,B 0,C 180,E1 -9926.492,E2 -9926.492} C_VEL
LIN {X 0,Y 425.255,Z 221.512,A -85,B 0,C 180,E1 -9929.714,E2 -9929.714} C_VEL
LIN {X 0,Y 425.245,Z 221.514,A -85,B 0,C 180,E1 -9933.043,E2 -9933.043} C_VEL
LIN {X 0,Y 425.242,Z 221.512,A -85,B 0,C 180,E1 -9935.923,E2 -9935.923} C_VEL
LIN {X 0,Y 425.254,Z 221.513,A -85,B 0,C 180,E1 -9939.038,E2 -9939.038} C_VEL
LIN {X 0,Y 425.233,Z 221.513,A -85,B 0,C 180,E1 -9942.648,E2 -9942.648} C_VEL
LIN {X 0,Y 425.214,Z 221.515,A -85,B 0,C 180,E1 -9946.039,E2 -9946.039} C_VEL
LIN {X 0,Y 425.224,Z 221.514,A -85,B 0,C 180,E1 -9948.617,E2 -9948.617} C_VEL
LIN {X 0,Y 425.258,Z 221.514,A -85,B 0,C 180,E1 -9951.098,E2 -9951.098} C_VEL
LIN {X 0,Y 425.247,Z 221.511,A -85,B 0,C 180,E1 -9954.66,E2 -9954.66} C_VEL
LIN {X 0,Y 425.21,Z 221.515,A -85,B 0,C 180,E1 -9958.069,E2 -9958.069} C_VEL
LIN {X 0,Y 425.281,Z 221.511,A -85,B 0,C 180,E1 -9961.365,E2 -9961.365} C_VEL
LIN {X 0,Y 425.242,Z 221.512,A -85,B 0,C 180,E1 -9964.552,E2 -9964.552} C_VEL
LIN {X 0,Y 425.264,Z 221.509,A -85,B 0,C 180,E1 -9967.716,E2 -9967.716} C_VEL
LIN {X 0,Y 425.305,Z 221.505,A -85,B 0,C 180,E1 -9970.702,E2 -9970.702} C_VEL
LIN {X 0,Y 425.337,Z 221.5,A -85,B 0,C 180,E1 -9973.687,E2 -9973.687} C_VEL
LIN {X 0,Y 425.369,Z 221.497,A -85,B 0,C 180,E1 -9977.597,E2 -9977.597} C_VEL
LIN {X 0,Y 425.403,Z 221.494,A -85,B 0,C 180,E1 -9981.449,E2 -9981.449} C_VEL
LIN {X 0,Y 425.521,Z 221.476,A -85,B 0,C 180,E1 -9984.313,E2 -9984.313} C_VEL
LIN {X 0,Y 425.512,Z 221.477,A -85,B 0,C 180,E1 -9988.107,E2 -9988.107} C_VEL
LIN {X 0,Y 425.64,Z 221.461,A -85,B 0,C 180,E1 -9990,E2 -9990} C_VEL
LIN {X 0,Y 425.502,Z 221.484,A -85,B 0,C 180,E1 -9992.84,E2 -9992.84} C_VEL
LIN {X 0,Y 425.521,Z 221.479,A -85,B 0,C 180,E1 -9995.687,E2 -9995.687} C_VEL
LIN {X 0,Y 425.404,Z 221.495,A -85,B 0,C 180,E1 -9998.551,E2 -9998.551} C_VEL
LIN {X 0,Y 425.359,Z 221.5,A -85,B 0,C 180,E1 -9999.105,E2 -9999.105} C_VEL
LIN {X 0,Y 424.689,Z 221.695,A -85,B 0,C 180,E1 -9999.641,E2 -9999.641} C_VEL
LIN {X 0,Y 421.983,Z 222.796,A -85,B 0,C 180,E1 -10000.478,E2 -10000.478} C_VEL
LIN {X 0,Y 419.851,Z 224.399,A -85,B 0,C 180,E1 -10001.126,E2 -10001.126} C_VEL
LIN {X 0,Y 419.092,Z 226.375,A -85,B 0,C 180,E1 -10001.695,E2 -10001.695} C_VEL
LIN {X 0,Y 419.131,Z 226.7,A -85,B 0,C 180,E1 -10001.775,E2 -10001.775} C_VEL
LIN {X 0,Y 420.009,Z 233.166,A -85,B 0,C 180,E1 -10003.301,E2 -10003.301} C_VEL
LIN {X 0,Y 419.893,Z 236.917,A -85,B 0,C 180,E1 -10004.127,E2 -10004.127} C_VEL
LIN {X 0,Y 423.817,Z 256.973,A -85,B 0,C 180,E1 -10004.666,E2 -10004.666} C_VEL
LIN {X 0,Y 422.645,Z 344.322,A -85,B 0,C 180,E1 -10006.211,E2 -10006.211} C_VEL
LIN {X 0,Y 422.24,Z 357.945,A -85,B 0,C 180,E1 -10006.654,E2 -10006.654} C_VEL
LIN {X 0,Y 421.786,Z 370.559,A -85,B 0,C 180,E1 -10007.265,E2 -10007.265} C_VEL
LIN {X 0,Y 421.209,Z 382.171,A -85,B 0,C 180,E1 -10008.027,E2 -10008.027} C_VEL
LIN {X 0,Y 420.511,Z 393.93,A -85,B 0,C 180,E1 -10009.02,E2 -10009.02} C_VEL
LIN {X 0,Y 419.893,Z 403.291,A -85,B 0,C 180,E1 -10010.003,E2 -10010.003} C_VEL
LIN {X 0,Y 419.195,Z 412.125,A -85,B 0,C 180,E1 -10011.128,E2 -10011.128} C_VEL
LIN {X 0,Y 418.595,Z 421.355,A -85,B 0,C 180,E1 -10012.591,E2 -10012.591} C_VEL
LIN {X 0,Y 418.067,Z 428.684,A -85,B 0,C 180,E1 -10014.034,E2 -10014.034} C_VEL
LIN {X 0,Y 417.683,Z 434.297,A -85,B 0,C 180,E1 -10015.408,E2 -10015.408} C_VEL
LIN {X 0,Y 417.396,Z 439.539,A -85,B 0,C 180,E1 -10017.04,E2 -10017.04} C_VEL
LIN {X 0,Y 417.169,Z 443.696,A -85,B 0,C 180,E1 -10018.85,E2 -10018.85} C_VEL
LIN {X 0,Y 416.946,Z 446.461,A -85,B 0,C 180,E1 -10020.739,E2 -10020.739} C_VEL
LIN {X 0,Y 416.896,Z 447.624,A -85,B 0,C 180,E1 -10022.645,E2 -10022.645} C_VEL
LIN {X 0,Y 416.897,Z 447.386,A -85,B 0,C 180,E1 -10024.321,E2 -10024.321} C_VEL
LIN {X 0,Y 417.012,Z 445.783,A -85,B 0,C 180,E1 -10026.146,E2 -10026.146} C_VEL
LIN {X 0,Y 417.241,Z 443.297,A -85,B 0,C 180,E1 -10027.672,E2 -10027.672} C_VEL
LIN {X 0,Y 417.437,Z 439.562,A -85,B 0,C 180,E1 -10029.257,E2 -10029.257} C_VEL
LIN {X 0,Y 417.797,Z 433.93,A -85,B 0,C 180,E1 -10030.997,E2 -10030.997} C_VEL
LIN {X 0,Y 418.301,Z 427.341,A -85,B 0,C 180,E1 -10032.566,E2 -10032.566} C_VEL
LIN {X 0,Y 418.89,Z 419.777,A -85,B 0,C 180,E1 -10033.995,E2 -10033.995} C_VEL
LIN {X 0,Y 419.653,Z 410.498,A -85,B 0,C 180,E1 -10035.397,E2 -10035.397} C_VEL
LIN {X 0,Y 420.312,Z 400.856,A -85,B 0,C 180,E1 -10036.58,E2 -10036.58} C_VEL
LIN {X 0,Y 421.061,Z 390.436,A -85,B 0,C 180,E1 -10037.608,E2 -10037.608} C_VEL
LIN {X 0,Y 421.83,Z 378.049,A -85,B 0,C 180,E1 -10038.565,E2 -10038.565} C_VEL
LIN {X 0,Y 422.411,Z 365.998,A -85,B 0,C 180,E1 -10039.278,E2 -10039.278} C_VEL
LIN {X 0,Y 422.874,Z 353.309,A -85,B 0,C 180,E1 -10039.813,E2 -10039.813} C_VEL
LIN {X 0,Y 423.192,Z 339.516,A -85,B 0,C 180,E1 -10040.18,E2 -10040.18} C_VEL
LIN {X 0,Y 424.32,Z 256.342,A -85,B 0,C 180,E1 -10041.65,E2 -10041.65} C_VEL
LIN {X 0,Y 420.173,Z 236.98,A -85,B 0,C 180,E1 -10042.219,E2 -10042.219} C_VEL
LIN {X 0,Y 420.101,Z 231.329,A -85,B 0,C 180,E1 -10043.416,E2 -10043.416} C_VEL
LIN {X 0,Y 418.266,Z 222.386,A -85,B 0,C 180,E1 -10045.465,E2 -10045.465} C_VEL
LIN {X 0,Y 418.209,Z 222.396,A -85,B 0,C 180,E1 -10048.985,E2 -10048.985} C_VEL
LIN {X 0,Y 418.262,Z 222.383,A -85,B 0,C 180,E1 -10051.943,E2 -10051.943} C_VEL
LIN {X 0,Y 418.26,Z 222.387,A -85,B 0,C 180,E1 -10055.168,E2 -10055.168} C_VEL
LIN {X 0,Y 418.205,Z 222.389,A -85,B 0,C 180,E1 -10058.309,E2 -10058.309} C_VEL
LIN {X 0,Y 418.258,Z 222.387,A -85,B 0,C 180,E1 -10061.389,E2 -10061.389} C_VEL
LIN {X 0,Y 418.279,Z 222.384,A -85,B 0,C 180,E1 -10064.412,E2 -10064.412} C_VEL
LIN {X 0,Y 418.35,Z 222.372,A -85,B 0,C 180,E1 -10067.392,E2 -10067.392} C_VEL
LIN {X 0,Y 418.325,Z 222.376,A -85,B 0,C 180,E1 -10070.334,E2 -10070.334} C_VEL
LIN {X 0,Y 418.454,Z 222.36,A -85,B 0,C 180,E1 -10073.254,E2 -10073.254} C_VEL
LIN {X 0,Y 418.318,Z 222.377,A -85,B 0,C 180,E1 -10075.187,E2 -10075.187} C_VEL
LIN {X 0,Y 418.529,Z 222.347,A -85,B 0,C 180,E1 -10078.081,E2 -10078.081} C_VEL
LIN {X 0,Y 418.655,Z 222.332,A -85,B 0,C 180,E1 -10080.005,E2 -10080.005} C_VEL
LIN {X 0,Y 418.467,Z 222.358,A -85,B 0,C 180,E1 -10082.893,E2 -10082.893} C_VEL
LIN {X 0,Y 418.491,Z 222.348,A -85,B 0,C 180,E1 -10085.788,E2 -10085.788} C_VEL
LIN {X 0,Y 418.369,Z 222.371,A -85,B 0,C 180,E1 -10088.701,E2 -10088.701} C_VEL
LIN {X 0,Y 418.307,Z 222.375,A -85,B 0,C 180,E1 -10091.636,E2 -10091.636} C_VEL
LIN {X 0,Y 418.298,Z 222.376,A -85,B 0,C 180,E1 -10094.602,E2 -10094.602} C_VEL
LIN {X 0,Y 418.278,Z 222.377,A -85,B 0,C 180,E1 -10097.609,E2 -10097.609} C_VEL
LIN {X 0,Y 418.25,Z 222.388,A -85,B 0,C 180,E1 -10100.668,E2 -10100.668} C_VEL
LIN {X 0,Y 418.255,Z 222.38,A -85,B 0,C 180,E1 -10103.788,E2 -10103.788} C_VEL
LIN {X 0,Y 418.204,Z 222.389,A -85,B 0,C 180,E1 -10107.045,E2 -10107.045} C_VEL
LIN {X 0,Y 418.243,Z 222.384,A -85,B 0,C 180,E1 -10110.277,E2 -10110.277} C_VEL
LIN {X 0,Y 418.235,Z 222.381,A -85,B 0,C 180,E1 -10113.683,E2 -10113.683} C_VEL
LIN {X 0,Y 418.237,Z 222.384,A -85,B 0,C 180,E1 -10117.229,E2 -10117.229} C_VEL
LIN {X 0,Y 418.212,Z 222.391,A -85,B 0,C 180,E1 -10120.953,E2 -10120.953} C_VEL
LIN {X 0,Y 418.198,Z 222.394,A -85,B 0,C 180,E1 -10123.729,E2 -10123.729} C_VEL
LIN {X 0,Y 418.185,Z 222.398,A -85,B 0,C 180,E1 -10126.447,E2 -10126.447} C_VEL
LIN {X 0,Y 418.214,Z 222.389,A -85,B 0,C 180,E1 -10129.136,E2 -10129.136} C_VEL
LIN {X 0,Y 418.239,Z 222.388,A -85,B 0,C 180,E1 -10132.777,E2 -10132.777} C_VEL
LIN {X 0,Y 418.236,Z 222.391,A -85,B 0,C 180,E1 -10136.323,E2 -10136.323} C_VEL
LIN {X 0,Y 418.244,Z 222.393,A -85,B 0,C 180,E1 -10139.729,E2 -10139.729} C_VEL
LIN {X 0,Y 418.24,Z 222.394,A -85,B 0,C 180,E1 -10142.319,E2 -10142.319} C_VEL
LIN {X 0,Y 420.753,Z 234.622,A -85,B 0,C 180,E1 -10144.936,E2 -10144.936} C_VEL
LIN {X 0,Y 421.257,Z 239.237,A -85,B 0,C 180,E1 -10145.875,E2 -10145.875} C_VEL
LIN {X 0,Y 420.221,Z 255.171,A -85,B 0,C 180,E1 -10148.926,E2 -10148.926} C_VEL
LIN {X 0,Y 419.701,Z 264.944,A -85,B 0,C 180,E1 -10150.784,E2 -10150.784} C_VEL
LIN {X 0,Y 423.835,Z 291.068,A -85,B 0,C 180,E1 -10151.481,E2 -10151.481} C_VEL
LIN {X 0,Y 422.934,Z 374.004,A -85,B 0,C 180,E1 -10152.97,E2 -10152.97} C_VEL
LIN {X 0,Y 422.36,Z 387.073,A -85,B 0,C 180,E1 -10153.382,E2 -10153.382} C_VEL
LIN {X 0,Y 421.685,Z 399.731,A -85,B 0,C 180,E1 -10153.977,E2 -10153.977} C_VEL
LIN {X 0,Y 420.928,Z 411.823,A -85,B 0,C 180,E1 -10154.754,E2 -10154.754} C_VEL
LIN {X 0,Y 420.192,Z 423.409,A -85,B 0,C 180,E1 -10155.722,E2 -10155.722} C_VEL
LIN {X 0,Y 419.409,Z 433.789,A -85,B 0,C 180,E1 -10156.803,E2 -10156.803} C_VEL
LIN {X 0,Y 418.848,Z 442.323,A -85,B 0,C 180,E1 -10157.893,E2 -10157.893} C_VEL
LIN {X 0,Y 418.073,Z 451.575,A -85,B 0,C 180,E1 -10159.344,E2 -10159.344} C_VEL
LIN {X 0,Y 417.645,Z 459.034,A -85,B 0,C 180,E1 -10160.801,E2 -10160.801} C_VEL
LIN {X 0,Y 417.339,Z 465.029,A -85,B 0,C 180,E1 -10162.258,E2 -10162.258} C_VEL
LIN {X 0,Y 417.126,Z 469.951,A -85,B 0,C 180,E1 -10163.775,E2 -10163.775} C_VEL
LIN {X 0,Y 417.108,Z 473.388,A -85,B 0,C 180,E1 -10165.167,E2 -10165.167} C_VEL
LIN {X 0,Y 417.02,Z 475.243,A -85,B 0,C 180,E1 -10166.135,E2 -10166.135} C_VEL
LIN {X 0,Y 417.036,Z 476.642,A -85,B 0,C 180,E1 -10167.102,E2 -10167.102} C_VEL
LIN {X 0,Y 417.076,Z 477.643,A -85,B 0,C 180,E1 -10168.069,E2 -10168.069} C_VEL
LIN {X 0,Y 417.02,Z 478.248,A -85,B 0,C 180,E1 -10169.034,E2 -10169.034} C_VEL
LIN {X 0,Y 417.012,Z 478.439,A -85,B 0,C 180,E1 -10170,E2 -10170} C_VEL
LIN {X 0,Y 417.076,Z 477.577,A -85,B 0,C 180,E1 -10171.931,E2 -10171.931} C_VEL
LIN {X 0,Y 417.037,Z 476.555,A -85,B 0,C 180,E1 -10172.898,E2 -10172.898} C_VEL
LIN {X 0,Y 417.02,Z 475.101,A -85,B 0,C 180,E1 -10173.865,E2 -10173.865} C_VEL
LIN {X 0,Y 417.097,Z 472.098,A -85,B 0,C 180,E1 -10175.317,E2 -10175.317} C_VEL
LIN {X 0,Y 417.243,Z 468.031,A -85,B 0,C 180,E1 -10176.771,E2 -10176.771} C_VEL
LIN {X 0,Y 417.499,Z 461.766,A -85,B 0,C 180,E1 -10178.47,E2 -10178.47} C_VEL
LIN {X 0,Y 417.868,Z 454.94,A -85,B 0,C 180,E1 -10179.927,E2 -10179.927} C_VEL
LIN {X 0,Y 418.416,Z 446.442,A -85,B 0,C 180,E1 -10181.382,E2 -10181.382} C_VEL
LIN {X 0,Y 419.033,Z 437.684,A -85,B 0,C 180,E1 -10182.593,E2 -10182.593} C_VEL
LIN {X 0,Y 419.726,Z 427.1,A -85,B 0,C 180,E1 -10183.783,E2 -10183.783} C_VEL
LIN {X 0,Y 420.404,Z 416.162,A -85,B 0,C 180,E1 -10184.77,E2 -10184.77} C_VEL
